LIN {X 0,Y 353.658,Z 542.313,A -85,B 0,C 180,E1 -13402.004,E2 -13402.004} C_VEL
LIN {X 0,Y 353.447,Z 546.534,A -85,B 0,C 180,E1 -13403.832,E2 -13403.832} C_VEL
LIN {X 0,Y 353.361,Z 549.292,A -85,B 0,C 180,E1 -13405.437,E2 -13405.437} C_VEL
LIN {X 0,Y 353.332,Z 551.715,A -85,B 0,C 180,E1 -13407.72,E2 -13407.72} C_VEL
LIN {X 0,Y 353.402,Z 552.336,A -85,B 0,C 180,E1 -13408.86,E2 -13408.86} C_VEL
LIN {X 0,Y 353.411,Z 552.555,A -85,B 0,C 180,E1 -13410,E2 -13410} C_VEL
LIN {X 0,Y 353.42,Z 552.336,A -85,B 0,C 180,E1 -13411.139,E2 -13411.139} C_VEL
LIN {X 0,Y 353.332,Z 551.714,A -85,B 0,C 180,E1 -13412.28,E2 -13412.28} C_VEL
LIN {X 0,Y 353.36,Z 549.289,A -85,B 0,C 180,E1 -13414.563,E2 -13414.563} C_VEL
LIN {X 0,Y 353.446,Z 546.529,A -85,B 0,C 180,E1 -13416.167,E2 -13416.167} C_VEL
LIN {X 0,Y 353.653,Z 542.299,A -85,B 0,C 180,E1 -13417.996,E2 -13417.996} C_VEL
LIN {X 0,Y 354.203,Z 536.136,A -85,B 0,C 180,E1 -13419.998,E2 -13419.998} C_VEL
LIN {X 0,Y 354.809,Z 529.405,A -85,B 0,C 180,E1 -13421.714,E2 -13421.714} C_VEL
LIN {X 0,Y 355.835,Z 521.078,A -85,B 0,C 180,E1 -13423.419,E2 -13423.419} C_VEL
LIN {X 0,Y 356.804,Z 512.544,A -85,B 0,C 180,E1 -13424.837,E2 -13424.837} C_VEL
LIN {X 0,Y 357.663,Z 503.178,A -85,B 0,C 180,E1 -13426.114,E2 -13426.114} C_VEL
LIN {X 0,Y 358.907,Z 491.587,A -85,B 0,C 180,E1 -13427.375,E2 -13427.375} C_VEL
LIN {X 0,Y 359.729,Z 483.732,A -85,B 0,C 180,E1 -13428.068,E2 -13428.068} C_VEL
LIN {X 0,Y 358.634,Z 471.661,A -85,B 0,C 180,E1 -13429.025,E2 -13429.025} C_VEL
LIN {X 0,Y 356.865,Z 458.288,A -85,B 0,C 180,E1 -13429.859,E2 -13429.859} C_VEL
LIN {X 0,Y 354.4,Z 444.565,A -85,B 0,C 180,E1 -13430.496,E2 -13430.496} C_VEL
LIN {X 0,Y 354.928,Z 437.738,A -85,B 0,C 180,E1 -13433.871,E2 -13433.871} C_VEL
LIN {X 0,Y 355.677,Z 429.964,A -85,B 0,C 180,E1 -13437.687,E2 -13437.687} C_VEL
LIN {X 0,Y 356.481,Z 422.367,A -85,B 0,C 180,E1 -13441.46,E2 -13441.46} C_VEL
LIN {X 0,Y 357.26,Z 415.856,A -85,B 0,C 180,E1 -13444.784,E2 -13444.784} C_VEL
LIN {X 0,Y 357.465,Z 411.958,A -85,B 0,C 180,E1 -13446.86,E2 -13446.86} C_VEL
LIN {X 0,Y 356.763,Z 406.874,A -85,B 0,C 180,E1 -13449.801,E2 -13449.801} C_VEL
LIN {X 0,Y 355.812,Z 401.617,A -85,B 0,C 180,E1 -13453.044,E2 -13453.044} C_VEL
LIN {X 0,Y 354.813,Z 396.295,A -85,B 0,C 180,E1 -13456.602,E2 -13456.602} C_VEL
LIN {X 0,Y 354.817,Z 396.29,A -85,B 0,C 180,E1 -13460.666,E2 -13460.666} C_VEL
LIN {X 0,Y 354.824,Z 396.285,A -85,B 0,C 180,E1 -13464.301,E2 -13464.301} C_VEL
LIN {X 0,Y 354.79,Z 396.288,A -85,B 0,C 180,E1 -13467.667,E2 -13467.667} C_VEL
LIN {X 0,Y 354.848,Z 396.28,A -85,B 0,C 180,E1 -13471.619,E2 -13471.619} C_VEL
LIN {X 0,Y 354.901,Z 396.275,A -85,B 0,C 180,E1 -13474.173,E2 -13474.173} C_VEL
LIN {X 0,Y 354.837,Z 396.282,A -85,B 0,C 180,E1 -13477.894,E2 -13477.894} C_VEL
LIN {X 0,Y 354.925,Z 396.271,A -85,B 0,C 180,E1 -13481.892,E2 -13481.892} C_VEL
LIN {X 0,Y 354.946,Z 396.269,A -85,B 0,C 180,E1 -13485.981,E2 -13485.981} C_VEL
LIN {X 0,Y 354.986,Z 396.263,A -85,B 0,C 180,E1 -13489.736,E2 -13489.736} C_VEL
LIN {X 0,Y 355.118,Z 396.249,A -85,B 0,C 180,E1 -13492.037,E2 -13492.037} C_VEL
LIN {X 0,Y 355.095,Z 396.255,A -85,B 0,C 180,E1 -13494.321,E2 -13494.321} C_VEL
LIN {X 0,Y 355.247,Z 396.231,A -85,B 0,C 180,E1 -13497.732,E2 -13497.732} C_VEL
LIN {X 0,Y 355.401,Z 396.214,A -85,B 0,C 180,E1 -13500,E2 -13500} C_VEL
LIN {X 0,Y 355.247,Z 396.236,A -85,B 0,C 180,E1 -13502.268,E2 -13502.268} C_VEL
LIN {X 0,Y 355.142,Z 396.245,A -85,B 0,C 180,E1 -13506.819,E2 -13506.819} C_VEL
LIN {X 0,Y 355.018,Z 396.259,A -85,B 0,C 180,E1 -13509.112,E2 -13509.112} C_VEL
LIN {X 0,Y 354.924,Z 396.273,A -85,B 0,C 180,E1 -13512.581,E2 -13512.581} C_VEL
LIN {X 0,Y 354.893,Z 396.281,A -85,B 0,C 180,E1 -13516.096,E2 -13516.096} C_VEL
LIN {X 0,Y 354.906,Z 396.275,A -85,B 0,C 180,E1 -13518.472,E2 -13518.472} C_VEL
LIN {X 0,Y 354.829,Z 396.288,A -85,B 0,C 180,E1 -13522.107,E2 -13522.107} C_VEL
LIN {X 0,Y 354.901,Z 396.278,A -85,B 0,C 180,E1 -13525.827,E2 -13525.827} C_VEL
LIN {X 0,Y 354.82,Z 396.287,A -85,B 0,C 180,E1 -13529.682,E2 -13529.682} C_VEL
LIN {X 0,Y 354.808,Z 396.289,A -85,B 0,C 180,E1 -13533.702,E2 -13533.702} C_VEL
LIN {X 0,Y 354.804,Z 396.286,A -85,B 0,C 180,E1 -13536.459,E2 -13536.459} C_VEL
LIN {X 0,Y 354.826,Z 396.286,A -85,B 0,C 180,E1 -13539.424,E2 -13539.424} C_VEL
LIN {X 0,Y 354.793,Z 396.287,A -85,B 0,C 180,E1 -13542.868,E2 -13542.868} C_VEL
LIN {X 0,Y 354.854,Z 396.281,A -85,B 0,C 180,E1 -13546.117,E2 -13546.117} C_VEL
LIN {X 0,Y 354.859,Z 396.281,A -85,B 0,C 180,E1 -13549.189,E2 -13549.189} C_VEL
LIN {X 0,Y 354.792,Z 396.288,A -85,B 0,C 180,E1 -13552.406,E2 -13552.406} C_VEL
LIN {X 0,Y 354.649,Z 396.307,A -85,B 0,C 180,E1 -13554.922,E2 -13554.922} C_VEL
LIN {X 0,Y 354.269,Z 396.37,A -85,B 0,C 180,E1 -13558.544,E2 -13558.544} C_VEL
LIN {X 0,Y 354.19,Z 398.943,A -85,B 0,C 180,E1 -13561.561,E2 -13561.561} C_VEL
LIN {X 0,Y 354.109,Z 401.198,A -85,B 0,C 180,E1 -13564.111,E2 -13564.111} C_VEL
LIN {X 0,Y 354.046,Z 403.503,A -85,B 0,C 180,E1 -13566.609,E2 -13566.609} C_VEL
LIN {X 0,Y 354.017,Z 406.555,A -85,B 0,C 180,E1 -13569.603,E2 -13569.603} C_VEL
LIN {X 0,Y 357.841,Z 419.612,A -85,B 0,C 180,E1 -13570.357,E2 -13570.357} C_VEL
LIN {X 0,Y 360.654,Z 431.525,A -85,B 0,C 180,E1 -13571.219,E2 -13571.219} C_VEL
LIN {X 0,Y 361.301,Z 435.514,A -85,B 0,C 180,E1 -13571.542,E2 -13571.542} C_VEL
LIN {X 0,Y 360.301,Z 447.888,A -85,B 0,C 180,E1 -13572.548,E2 -13572.548} C_VEL
LIN {X 0,Y 359.4,Z 458.522,A -85,B 0,C 180,E1 -13573.674,E2 -13573.674} C_VEL
LIN {X 0,Y 358.359,Z 468.201,A -85,B 0,C 180,E1 -13574.939,E2 -13574.939} C_VEL
LIN {X 0,Y 357.248,Z 477.008,A -85,B 0,C 180,E1 -13576.345,E2 -13576.345} C_VEL
LIN {X 0,Y 356.228,Z 485.588,A -85,B 0,C 180,E1 -13578.044,E2 -13578.044} C_VEL
LIN {X 0,Y 355.358,Z 492.423,A -85,B 0,C 180,E1 -13579.747,E2 -13579.747} C_VEL
LIN {X 0,Y 354.706,Z 497.89,A -85,B 0,C 180,E1 -13581.454,E2 -13581.454} C_VEL
LIN {X 0,Y 354.252,Z 502.177,A -85,B 0,C 180,E1 -13583.164,E2 -13583.164} C_VEL
LIN {X 0,Y 353.919,Z 504.45,A -85,B 0,C 180,E1 -13584.302,E2 -13584.302} C_VEL
LIN {X 0,Y 353.78,Z 506.291,A -85,B 0,C 180,E1 -13585.442,E2 -13585.442} C_VEL
LIN {X 0,Y 353.784,Z 507.67,A -85,B 0,C 180,E1 -13586.583,E2 -13586.583} C_VEL
LIN {X 0,Y 353.508,Z 509.272,A -85,B 0,C 180,E1 -13588.861,E2 -13588.861} C_VEL
LIN {X 0,Y 353.477,Z 509.503,A -85,B 0,C 180,E1 -13590,E2 -13590} C_VEL
LIN {X 0,Y 353.636,Z 508.728,A -85,B 0,C 180,E1 -13592.278,E2 -13592.278} C_VEL
LIN {X 0,Y 353.764,Z 507.766,A -85,B 0,C 180,E1 -13593.417,E2 -13593.417} C_VEL
LIN {X 0,Y 353.777,Z 506.428,A -85,B 0,C 180,E1 -13594.558,E2 -13594.558} C_VEL
LIN {X 0,Y 354.082,Z 503.581,A -85,B 0,C 180,E1 -13596.267,E2 -13596.267} C_VEL
LIN {X 0,Y 354.483,Z 499.722,A -85,B 0,C 180,E1 -13597.978,E2 -13597.978} C_VEL
LIN {X 0,Y 355.096,Z 494.736,A -85,B 0,C 180,E1 -13599.685,E2 -13599.685} C_VEL
LIN {X 0,Y 355.914,Z 488.452,A -85,B 0,C 180,E1 -13601.389,E2 -13601.389} C_VEL
LIN {X 0,Y 356.891,Z 480.584,A -85,B 0,C 180,E1 -13603.089,E2 -13603.089} C_VEL
LIN {X 0,Y 357.857,Z 472.558,A -85,B 0,C 180,E1 -13604.501,E2 -13604.501} C_VEL
LIN {X 0,Y 358.974,Z 462.756,A -85,B 0,C 180,E1 -13605.908,E2 -13605.908} C_VEL
LIN {X 0,Y 359.828,Z 453.112,A -85,B 0,C 180,E1 -13607.036,E2 -13607.036} C_VEL
LIN {X 0,Y 360.762,Z 442.655,A -85,B 0,C 180,E1 -13608.015,E2 -13608.015} C_VEL
LIN {X 0,Y 361.217,Z 433.881,A -85,B 0,C 180,E1 -13608.687,E2 -13608.687} C_VEL
LIN {X 0,Y 358.725,Z 422.991,A -85,B 0,C 180,E1 -13609.522,E2 -13609.522} C_VEL
LIN {X 0,Y 355.128,Z 410.483,A -85,B 0,C 180,E1 -13610.301,E2 -13610.301} C_VEL
LIN {X 0,Y 353.959,Z 406.397,A -85,B 0,C 180,E1 -13610.514,E2 -13610.514} C_VEL
LIN {X 0,Y 354.101,Z 402.965,A -85,B 0,C 180,E1 -13614.078,E2 -13614.078} C_VEL
LIN {X 0,Y 354.141,Z 400.17,A -85,B 0,C 180,E1 -13617.158,E2 -13617.158} C_VEL
LIN {X 0,Y 354.258,Z 397.914,A -85,B 0,C 180,E1 -13619.734,E2 -13619.734} C_VEL
LIN {X 0,Y 354.3,Z 396.464,A -85,B 0,C 180,E1 -13621.464,E2 -13621.464} C_VEL
LIN {X 0,Y 354.651,Z 396.307,A -85,B 0,C 180,E1 -13625.078,E2 -13625.078} C_VEL
LIN {X 0,Y 354.769,Z 396.29,A -85,B 0,C 180,E1 -13627.355,E2 -13627.355} C_VEL
LIN {X 0,Y 354.164,Z 396.37,A -85,B 0,C 180,E1 -13628.302,E2 -13628.302} C_VEL
LIN {X 0,Y 351.329,Z 396.72,A -85,B 0,C 180,E1 -13629.843,E2 -13629.843} C_VEL
LIN {X 0,Y 348.879,Z 397.025,A -85,B 0,C 180,E1 -13631.09,E2 -13631.09} C_VEL
LIN {X 0,Y 347.811,Z 397.159,A -85,B 0,C 180,E1 -13632.055,E2 -13632.055} C_VEL
LIN {X 0,Y 347.717,Z 397.166,A -85,B 0,C 180,E1 -13632.382,E2 -13632.382} C_VEL
LIN {X 0,Y 347.709,Z 397.17,A -85,B 0,C 180,E1 -13635.027,E2 -13635.027} C_VEL
LIN {X 0,Y 347.754,Z 397.17,A -85,B 0,C 180,E1 -13638.397,E2 -13638.397} C_VEL
LIN {X 0,Y 347.781,Z 397.164,A -85,B 0,C 180,E1 -13642.011,E2 -13642.011} C_VEL
LIN {X 0,Y 347.748,Z 397.165,A -85,B 0,C 180,E1 -13645.536,E2 -13645.536} C_VEL
LIN {X 0,Y 347.749,Z 397.17,A -85,B 0,C 180,E1 -13648.301,E2 -13648.301} C_VEL
LIN {X 0,Y 347.782,Z 397.161,A -85,B 0,C 180,E1 -13650.988,E2 -13650.988} C_VEL
LIN {X 0,Y 347.834,Z 397.156,A -85,B 0,C 180,E1 -13653.608,E2 -13653.608} C_VEL
LIN {X 0,Y 347.789,Z 397.165,A -85,B 0,C 180,E1 -13656.162,E2 -13656.162} C_VEL
LIN {X 0,Y 347.813,Z 397.162,A -85,B 0,C 180,E1 -13659.909,E2 -13659.909} C_VEL
LIN {X 0,Y 347.87,Z 397.152,A -85,B 0,C 180,E1 -13662.359,E2 -13662.359} C_VEL
LIN {X 0,Y 347.901,Z 397.151,A -85,B 0,C 180,E1 -13665.971,E2 -13665.971} C_VEL
LIN {X 0,Y 347.931,Z 397.145,A -85,B 0,C 180,E1 -13669.526,E2 -13669.526} C_VEL
LIN {X 0,Y 348.084,Z 397.123,A -85,B 0,C 180,E1 -13673.042,E2 -13673.042} C_VEL
LIN {X 0,Y 348.21,Z 397.113,A -85,B 0,C 180,E1 -13677.686,E2 -13677.686} C_VEL
LIN {X 0,Y 348.349,Z 397.093,A -85,B 0,C 180,E1 -13680,E2 -13680} C_VEL
LIN {X 0,Y 348.21,Z 397.108,A -85,B 0,C 180,E1 -13682.313,E2 -13682.313} C_VEL
LIN {X 0,Y 348.111,Z 397.12,A -85,B 0,C 180,E1 -13686.958,E2 -13686.958} C_VEL
LIN {X 0,Y 347.973,Z 397.14,A -85,B 0,C 180,E1 -13689.298,E2 -13689.298} C_VEL
LIN {X 0,Y 347.898,Z 397.147,A -85,B 0,C 180,E1 -13692.839,E2 -13692.839} C_VEL
LIN {X 0,Y 347.843,Z 397.153,A -85,B 0,C 180,E1 -13696.431,E2 -13696.431} C_VEL
LIN {X 0,Y 347.855,Z 397.153,A -85,B 0,C 180,E1 -13698.86,E2 -13698.86} C_VEL
LIN {X 0,Y 347.778,Z 397.161,A -85,B 0,C 180,E1 -13702.579,E2 -13702.579} C_VEL
LIN {X 0,Y 347.816,Z 397.161,A -85,B 0,C 180,E1 -13705.108,E2 -13705.108} C_VEL
LIN {X 0,Y 347.811,Z 397.159,A -85,B 0,C 180,E1 -13707.694,E2 -13707.694} C_VEL
LIN {X 0,Y 347.752,Z 397.165,A -85,B 0,C 180,E1 -13710.348,E2 -13710.348} C_VEL
LIN {X 0,Y 347.751,Z 397.165,A -85,B 0,C 180,E1 -13714.044,E2 -13714.044} C_VEL
LIN {X 0,Y 347.765,Z 397.167,A -85,B 0,C 180,E1 -13717.32,E2 -13717.32} C_VEL
LIN {X 0,Y 347.735,Z 397.169,A -85,B 0,C 180,E1 -13720.297,E2 -13720.297} C_VEL
LIN {X 0,Y 347.773,Z 397.235,A -85,B 0,C 180,E1 -13722.971,E2 -13722.971} C_VEL
LIN {X 0,Y 348.737,Z 402.423,A -85,B 0,C 180,E1 -13726.511,E2 -13726.511} C_VEL
LIN {X 0,Y 349.739,Z 407.928,A -85,B 0,C 180,E1 -13729.981,E2 -13729.981} C_VEL
LIN {X 0,Y 350.471,Z 413.076,A -85,B 0,C 180,E1 -13733.016,E2 -13733.016} C_VEL
LIN {X 0,Y 350.197,Z 417.38,A -85,B 0,C 180,E1 -13735.368,E2 -13735.368} C_VEL
LIN {X 0,Y 349.43,Z 423.299,A -85,B 0,C 180,E1 -13738.471,E2 -13738.471} C_VEL
LIN {X 0,Y 348.601,Z 430.928,A -85,B 0,C 180,E1 -13742.374,E2 -13742.374} C_VEL
LIN {X 0,Y 347.838,Z 438.435,A -85,B 0,C 180,E1 -13746.165,E2 -13746.165} C_VEL
LIN {X 0,Y 347.377,Z 444.195,A -85,B 0,C 180,E1 -13749.071,E2 -13749.071} C_VEL
LIN {X 0,Y 349.885,Z 457.827,A -85,B 0,C 180,E1 -13749.719,E2 -13749.719} C_VEL
LIN {X 0,Y 351.588,Z 470.563,A -85,B 0,C 180,E1 -13750.528,E2 -13750.528} C_VEL
LIN {X 0,Y 352.829,Z 483.366,A -85,B 0,C 180,E1 -13751.566,E2 -13751.566} C_VEL
LIN {X 0,Y 351.846,Z 494.074,A -85,B 0,C 180,E1 -13752.565,E2 -13752.565} C_VEL
LIN {X 0,Y 350.581,Z 505.021,A -85,B 0,C 180,E1 -13753.851,E2 -13753.851} C_VEL
LIN {X 0,Y 349.688,Z 513.954,A -85,B 0,C 180,E1 -13755.152,E2 -13755.152} C_VEL
LIN {X 0,Y 348.731,Z 522.173,A -85,B 0,C 180,E1 -13756.599,E2 -13756.599} C_VEL
LIN {X 0,Y 347.667,Z 530.237,A -85,B 0,C 180,E1 -13758.337,E2 -13758.337} C_VEL
LIN {X 0,Y 347.071,Z 536.725,A -85,B 0,C 180,E1 -13760.089,E2 -13760.089} C_VEL
LIN {X 0,Y 346.595,Z 541.879,A -85,B 0,C 180,E1 -13761.84,E2 -13761.84} C_VEL
LIN {X 0,Y 346.344,Z 546.435,A -85,B 0,C 180,E1 -13763.885,E2 -13763.885} C_VEL
LIN {X 0,Y 346.275,Z 548.86,A -85,B 0,C 180,E1 -13765.343,E2 -13765.343} C_VEL
LIN {X 0,Y 346.237,Z 551.283,A -85,B 0,C 180,E1 -13767.673,E2 -13767.673} C_VEL
LIN {X 0,Y 346.322,Z 551.905,A -85,B 0,C 180,E1 -13768.837,E2 -13768.837} C_VEL
LIN {X 0,Y 346.35,Z 552.125,A -85,B 0,C 180,E1 -13770,E2 -13770} C_VEL
LIN {X 0,Y 346.339,Z 551.904,A -85,B 0,C 180,E1 -13771.163,E2 -13771.163} C_VEL
LIN {X 0,Y 346.206,Z 550.269,A -85,B 0,C 180,E1 -13773.491,E2 -13773.491} C_VEL
LIN {X 0,Y 346.274,Z 548.856,A -85,B 0,C 180,E1 -13774.657,E2 -13774.657} C_VEL
LIN {X 0,Y 346.343,Z 546.429,A -85,B 0,C 180,E1 -13776.113,E2 -13776.113} C_VEL
LIN {X 0,Y 346.591,Z 541.863,A -85,B 0,C 180,E1 -13778.16,E2 -13778.16} C_VEL
LIN {X 0,Y 347.171,Z 535.699,A -85,B 0,C 180,E1 -13780.203,E2 -13780.203} C_VEL
LIN {X 0,Y 347.819,Z 528.968,A -85,B 0,C 180,E1 -13781.953,E2 -13781.953} C_VEL
LIN {X 0,Y 348.865,Z 520.639,A -85,B 0,C 180,E1 -13783.692,E2 -13783.692} C_VEL
LIN {X 0,Y 349.932,Z 511.43,A -85,B 0,C 180,E1 -13785.238,E2 -13785.238} C_VEL
LIN {X 0,Y 350.949,Z 501.56,A -85,B 0,C 180,E1 -13786.581,E2 -13786.581} C_VEL
LIN {X 0,Y 352.282,Z 489.717,A -85,B 0,C 180,E1 -13787.862,E2 -13787.862} C_VEL
LIN {X 0,Y 352.82,Z 483.284,A -85,B 0,C 180,E1 -13788.435,E2 -13788.435} C_VEL
LIN {X 0,Y 351.587,Z 470.464,A -85,B 0,C 180,E1 -13789.47,E2 -13789.47} C_VEL
LIN {X 0,Y 349.733,Z 457.055,A -85,B 0,C 180,E1 -13790.316,E2 -13790.316} C_VEL
LIN {X 0,Y 347.391,Z 444.134,A -85,B 0,C 180,E1 -13790.919,E2 -13790.919} C_VEL
LIN {X 0,Y 348.085,Z 435.921,A -85,B 0,C 180,E1 -13795.087,E2 -13795.087} C_VEL
LIN {X 0,Y 348.873,Z 428.36,A -85,B 0,C 180,E1 -13798.913,E2 -13798.913} C_VEL
LIN {X 0,Y 349.762,Z 420.671,A -85,B 0,C 180,E1 -13802.856,E2 -13802.856} C_VEL
LIN {X 0,Y 350.378,Z 415.533,A -85,B 0,C 180,E1 -13805.57,E2 -13805.57} C_VEL
LIN {X 0,Y 350.334,Z 411.671,A -85,B 0,C 180,E1 -13807.724,E2 -13807.724} C_VEL
LIN {X 0,Y 349.526,Z 406.519,A -85,B 0,C 180,E1 -13810.835,E2 -13810.835} C_VEL
LIN {X 0,Y 348.533,Z 401.184,A -85,B 0,C 180,E1 -13814.279,E2 -13814.279} C_VEL
LIN {X 0,Y 347.75,Z 397.175,A -85,B 0,C 180,E1 -13817.122,E2 -13817.122} C_VEL
LIN {X 0,Y 347.754,Z 397.168,A -85,B 0,C 180,E1 -13821.208,E2 -13821.208} C_VEL
LIN {X 0,Y 347.791,Z 397.16,A -85,B 0,C 180,E1 -13824.125,E2 -13824.125} C_VEL
LIN {X 0,Y 347.741,Z 397.167,A -85,B 0,C 180,E1 -13828.086,E2 -13828.086} C_VEL
LIN {X 0,Y 347.781,Z 397.165,A -85,B 0,C 180,E1 -13830.988,E2 -13830.988} C_VEL
LIN {X 0,Y 347.833,Z 397.154,A -85,B 0,C 180,E1 -13833.608,E2 -13833.608} C_VEL
LIN {X 0,Y 347.791,Z 397.161,A -85,B 0,C 180,E1 -13836.162,E2 -13836.162} C_VEL
LIN {X 0,Y 347.815,Z 397.157,A -85,B 0,C 180,E1 -13839.909,E2 -13839.909} C_VEL
LIN {X 0,Y 347.869,Z 397.153,A -85,B 0,C 180,E1 -13842.359,E2 -13842.359} C_VEL
LIN {X 0,Y 347.9,Z 397.147,A -85,B 0,C 180,E1 -13845.971,E2 -13845.971} C_VEL
LIN {X 0,Y 347.936,Z 397.141,A -85,B 0,C 180,E1 -13849.526,E2 -13849.526} C_VEL
LIN {X 0,Y 348.078,Z 397.125,A -85,B 0,C 180,E1 -13851.875,E2 -13851.875} C_VEL
LIN {X 0,Y 348.07,Z 397.129,A -85,B 0,C 180,E1 -13854.206,E2 -13854.206} C_VEL
LIN {X 0,Y 348.209,Z 397.108,A -85,B 0,C 180,E1 -13857.687,E2 -13857.687} C_VEL
LIN {X 0,Y 348.371,Z 397.09,A -85,B 0,C 180,E1 -13860,E2 -13860} C_VEL
LIN {X 0,Y 348.209,Z 397.113,A -85,B 0,C 180,E1 -13862.314,E2 -13862.314} C_VEL
LIN {X 0,Y 348.11,Z 397.12,A -85,B 0,C 180,E1 -13866.958,E2 -13866.958} C_VEL
LIN {X 0,Y 347.97,Z 397.137,A -85,B 0,C 180,E1 -13869.299,E2 -13869.299} C_VEL
LIN {X 0,Y 347.893,Z 397.147,A -85,B 0,C 180,E1 -13872.839,E2 -13872.839} C_VEL
LIN {X 0,Y 347.842,Z 397.156,A -85,B 0,C 180,E1 -13876.431,E2 -13876.431} C_VEL
LIN {X 0,Y 347.855,Z 397.151,A -85,B 0,C 180,E1 -13878.86,E2 -13878.86} C_VEL
LIN {X 0,Y 347.771,Z 397.163,A -85,B 0,C 180,E1 -13882.58,E2 -13882.58} C_VEL
LIN {X 0,Y 347.813,Z 397.157,A -85,B 0,C 180,E1 -13885.108,E2 -13885.108} C_VEL
LIN {X 0,Y 347.811,Z 397.16,A -85,B 0,C 180,E1 -13887.694,E2 -13887.694} C_VEL
LIN {X 0,Y 347.751,Z 397.166,A -85,B 0,C 180,E1 -13890.348,E2 -13890.348} C_VEL
LIN {X 0,Y 347.75,Z 397.169,A -85,B 0,C 180,E1 -13894.044,E2 -13894.044} C_VEL
LIN {X 0,Y 347.768,Z 397.163,A -85,B 0,C 180,E1 -13897.32,E2 -13897.32} C_VEL
LIN {X 0,Y 347.735,Z 397.168,A -85,B 0,C 180,E1 -13900.297,E2 -13900.297} C_VEL
LIN {X 0,Y 347.731,Z 397.17,A -85,B 0,C 180,E1 -13903.407,E2 -13903.407} C_VEL
LIN {X 0,Y 347.788,Z 397.16,A -85,B 0,C 180,E1 -13906.676,E2 -13906.676} C_VEL
LIN {X 0,Y 347.788,Z 397.161,A -85,B 0,C 180,E1 -13910.165,E2 -13910.165} C_VEL
LIN {X 0,Y 347.739,Z 397.167,A -85,B 0,C 180,E1 -13912.676,E2 -13912.676} C_VEL
LIN {X 0,Y 347.491,Z 397.202,A -85,B 0,C 180,E1 -13916.02,E2 -13916.02} C_VEL
LIN {X 0,Y 347.269,Z 397.229,A -85,B 0,C 180,E1 -13918.252,E2 -13918.252} C_VEL
LIN {X 0,Y 347.183,Z 399.317,A -85,B 0,C 180,E1 -13920.933,E2 -13920.933} C_VEL
LIN {X 0,Y 347.093,Z 401.598,A -85,B 0,C 180,E1 -13923.547,E2 -13923.547} C_VEL
LIN {X 0,Y 347.043,Z 403.914,A -85,B 0,C 180,E1 -13926.107,E2 -13926.107} C_VEL
LIN {X 0,Y 346.988,Z 406.939,A -85,B 0,C 180,E1 -13929.168,E2 -13929.168} C_VEL
LIN {X 0,Y 350.853,Z 420.05,A -85,B 0,C 180,E1 -13929.948,E2 -13929.948} C_VEL
LIN {X 0,Y 353.848,Z 432.487,A -85,B 0,C 180,E1 -13930.878,E2 -13930.878} C_VEL
LIN {X 0,Y 354.574,Z 436.195,A -85,B 0,C 180,E1 -13931.198,E2 -13931.198} C_VEL
LIN {X 0,Y 353.563,Z 448.324,A -85,B 0,C 180,E1 -13932.205,E2 -13932.205} C_VEL
LIN {X 0,Y 352.559,Z 459.427,A -85,B 0,C 180,E1 -13933.409,E2 -13933.409} C_VEL
LIN {X 0,Y 351.531,Z 468.635,A -85,B 0,C 180,E1 -13934.639,E2 -13934.639} C_VEL
LIN {X 0,Y 350.362,Z 477.443,A -85,B 0,C 180,E1 -13936.072,E2 -13936.072} C_VEL
LIN {X 0,Y 349.304,Z 486.021,A -85,B 0,C 180,E1 -13937.804,E2 -13937.804} C_VEL
LIN {X 0,Y 348.396,Z 492.856,A -85,B 0,C 180,E1 -13939.54,E2 -13939.54} C_VEL
LIN {X 0,Y 347.693,Z 498.324,A -85,B 0,C 180,E1 -13941.28,E2 -13941.28} C_VEL
LIN {X 0,Y 347.212,Z 502.61,A -85,B 0,C 180,E1 -13943.024,E2 -13943.024} C_VEL
LIN {X 0,Y 346.885,Z 504.882,A -85,B 0,C 180,E1 -13944.186,E2 -13944.186} C_VEL
LIN {X 0,Y 346.707,Z 506.724,A -85,B 0,C 180,E1 -13945.349,E2 -13945.349} C_VEL
LIN {X 0,Y 346.713,Z 508.102,A -85,B 0,C 180,E1 -13946.514,E2 -13946.514} C_VEL
LIN {X 0,Y 346.583,Z 509.09,A -85,B 0,C 180,E1 -13947.676,E2 -13947.676} C_VEL
LIN {X 0,Y 346.413,Z 509.933,A -85,B 0,C 180,E1 -13950,E2 -13950} C_VEL
LIN {X 0,Y 346.58,Z 509.158,A -85,B 0,C 180,E1 -13952.324,E2 -13952.324} C_VEL
LIN {X 0,Y 346.695,Z 508.197,A -85,B 0,C 180,E1 -13953.487,E2 -13953.487} C_VEL
LIN {X 0,Y 346.705,Z 506.859,A -85,B 0,C 180,E1 -13954.651,E2 -13954.651} C_VEL
LIN {X 0,Y 347.059,Z 504.011,A -85,B 0,C 180,E1 -13956.395,E2 -13956.395} C_VEL
LIN {X 0,Y 347.467,Z 500.152,A -85,B 0,C 180,E1 -13958.14,E2 -13958.14} C_VEL
LIN {X 0,Y 348.099,Z 495.167,A -85,B 0,C 180,E1 -13959.882,E2 -13959.882} C_VEL
LIN {X 0,Y 348.965,Z 488.882,A -85,B 0,C 180,E1 -13961.619,E2 -13961.619} C_VEL
LIN {X 0,Y 350.002,Z 481.012,A -85,B 0,C 180,E1 -13963.351,E2 -13963.351} C_VEL
LIN {X 0,Y 351.013,Z 472.985,A -85,B 0,C 180,E1 -13964.79,E2 -13964.79} C_VEL
LIN {X 0,Y 352.165,Z 463.183,A -85,B 0,C 180,E1 -13966.224,E2 -13966.224} C_VEL
LIN {X 0,Y 353.067,Z 453.538,A -85,B 0,C 180,E1 -13967.373,E2 -13967.373} C_VEL
LIN {X 0,Y 354.05,Z 443.078,A -85,B 0,C 180,E1 -13968.369,E2 -13968.369} C_VEL
LIN {X 0,Y 354.548,Z 435.819,A -85,B 0,C 180,E1 -13968.937,E2 -13968.937} C_VEL
LIN {X 0,Y 352.026,Z 424.588,A -85,B 0,C 180,E1 -13969.84,E2 -13969.84} C_VEL
LIN {X 0,Y 348.492,Z 412.001,A -85,B 0,C 180,E1 -13970.667,E2 -13970.667} C_VEL
LIN {X 0,Y 346.913,Z 406.812,A -85,B 0,C 180,E1 -13970.969,E2 -13970.969} C_VEL
LIN {X 0,Y 347.042,Z 403.633,A -85,B 0,C 180,E1 -13974.313,E2 -13974.313} C_VEL
LIN {X 0,Y 347.105,Z 400.558,A -85,B 0,C 180,E1 -13977.755,E2 -13977.755} C_VEL
LIN {X 0,Y 347.221,Z 398.286,A -85,B 0,C 180,E1 -13980.399,E2 -13980.399} C_VEL
LIN {X 0,Y 347.273,Z 397.23,A -85,B 0,C 180,E1 -13981.79,E2 -13981.79} C_VEL
LIN {X 0,Y 347.556,Z 397.195,A -85,B 0,C 180,E1 -13984.486,E2 -13984.486} C_VEL
LIN {X 0,Y 347.766,Z 397.164,A -85,B 0,C 180,E1 -13987.987,E2 -13987.987} C_VEL
LIN {X 0,Y 347.754,Z 397.165,A -85,B 0,C 180,E1 -13991.83,E2 -13991.83} C_VEL
LIN {X 0,Y 347.717,Z 397.166,A -85,B 0,C 180,E1 -13992.382,E2 -13992.382} C_VEL
LIN {X 0,Y 347.029,Z 397.255,A -85,B 0,C 180,E1 -13993.349,E2 -13993.349} C_VEL
LIN {X 0,Y 344.166,Z 397.612,A -85,B 0,C 180,E1 -13994.921,E2 -13994.921} C_VEL
LIN {X 0,Y 341.765,Z 397.914,A -85,B 0,C 180,E1 -13996.194,E2 -13996.194} C_VEL
LIN {X 0,Y 340.754,Z 398.036,A -85,B 0,C 180,E1 -13997.18,E2 -13997.18} C_VEL
LIN {X 0,Y 340.681,Z 398.045,A -85,B 0,C 180,E1 -13997.513,E2 -13997.513} C_VEL
LIN {X 0,Y 340.703,Z 398.048,A -85,B 0,C 180,E1 -14000.248,E2 -14000.248} C_VEL
LIN {X 0,Y 340.715,Z 398.041,A -85,B 0,C 180,E1 -14003.559,E2 -14003.559} C_VEL
LIN {X 0,Y 340.698,Z 398.048,A -85,B 0,C 180,E1 -14006.154,E2 -14006.154} C_VEL
LIN {X 0,Y 340.745,Z 398.041,A -85,B 0,C 180,E1 -14010.329,E2 -14010.329} C_VEL
LIN {X 0,Y 340.807,Z 398.029,A -85,B 0,C 180,E1 -14013.02,E2 -14013.02} C_VEL
LIN {X 0,Y 340.758,Z 398.037,A -85,B 0,C 180,E1 -14015.638,E2 -14015.638} C_VEL
LIN {X 0,Y 340.739,Z 398.039,A -85,B 0,C 180,E1 -14019.474,E2 -14019.474} C_VEL
LIN {X 0,Y 340.862,Z 398.029,A -85,B 0,C 180,E1 -14021.984,E2 -14021.984} C_VEL
LIN {X 0,Y 340.873,Z 398.025,A -85,B 0,C 180,E1 -14025.705,E2 -14025.705} C_VEL
LIN {X 0,Y 340.874,Z 398.022,A -85,B 0,C 180,E1 -14029.306,E2 -14029.306} C_VEL
LIN {X 0,Y 341.051,Z 397.999,A -85,B 0,C 180,E1 -14032.898,E2 -14032.898} C_VEL
LIN {X 0,Y 341.172,Z 397.99,A -85,B 0,C 180,E1 -14037.639,E2 -14037.639} C_VEL
LIN {X 0,Y 341.299,Z 397.972,A -85,B 0,C 180,E1 -14040,E2 -14040} C_VEL
LIN {X 0,Y 341.172,Z 397.985,A -85,B 0,C 180,E1 -14042.361,E2 -14042.361} C_VEL
LIN {X 0,Y 341.081,Z 397.997,A -85,B 0,C 180,E1 -14047.102,E2 -14047.102} C_VEL
LIN {X 0,Y 340.88,Z 398.021,A -85,B 0,C 180,E1 -14050.693,E2 -14050.693} C_VEL
LIN {X 0,Y 340.867,Z 398.022,A -85,B 0,C 180,E1 -14054.325,E2 -14054.325} C_VEL
LIN {X 0,Y 340.841,Z 398.025,A -85,B 0,C 180,E1 -14058.466,E2 -14058.466} C_VEL
LIN {X 0,Y 340.757,Z 398.037,A -85,B 0,C 180,E1 -14061.857,E2 -14061.857} C_VEL
LIN {X 0,Y 340.776,Z 398.036,A -85,B 0,C 180,E1 -14065.664,E2 -14065.664} C_VEL
LIN {X 0,Y 340.732,Z 398.039,A -85,B 0,C 180,E1 -14068.321,E2 -14068.321} C_VEL
LIN {X 0,Y 340.701,Z 398.048,A -85,B 0,C 180,E1 -14071.044,E2 -14071.044} C_VEL
LIN {X 0,Y 340.721,Z 398.044,A -85,B 0,C 180,E1 -14075.279,E2 -14075.279} C_VEL
LIN {X 0,Y 340.713,Z 398.044,A -85,B 0,C 180,E1 -14078.386,E2 -14078.386} C_VEL
LIN {X 0,Y 340.748,Z 398.17,A -85,B 0,C 180,E1 -14082.535,E2 -14082.535} C_VEL
LIN {X 0,Y 341.682,Z 403.184,A -85,B 0,C 180,E1 -14086.047,E2 -14086.047} C_VEL
LIN {X 0,Y 342.617,Z 408.296,A -85,B 0,C 180,E1 -14089.374,E2 -14089.374} C_VEL
LIN {X 0,Y 343.328,Z 412.759,A -85,B 0,C 180,E1 -14092.112,E2 -14092.112} C_VEL
LIN {X 0,Y 343.38,Z 416.594,A -85,B 0,C 180,E1 -14094.316,E2 -14094.316} C_VEL
LIN {X 0,Y 342.565,Z 422.956,A -85,B 0,C 180,E1 -14097.763,E2 -14097.763} C_VEL
LIN {X 0,Y 341.679,Z 430.549,A -85,B 0,C 180,E1 -14101.765,E2 -14101.765} C_VEL
LIN {X 0,Y 340.863,Z 438.03,A -85,B 0,C 180,E1 -14105.646,E2 -14105.646} C_VEL
LIN {X 0,Y 340.391,Z 443.766,A -85,B 0,C 180,E1 -14108.62,E2 -14108.62} C_VEL
LIN {X 0,Y 342.98,Z 457.807,A -85,B 0,C 180,E1 -14109.313,E2 -14109.313} C_VEL
LIN {X 0,Y 344.762,Z 471.402,A -85,B 0,C 180,E1 -14110.213,E2 -14110.213} C_VEL
LIN {X 0,Y 345.869,Z 482.924,A -85,B 0,C 180,E1 -14111.181,E2 -14111.181} C_VEL
LIN {X 0,Y 345.543,Z 489.353,A -85,B 0,C 180,E1 -14111.777,E2 -14111.777} C_VEL
LIN {X 0,Y 344.125,Z 501.183,A -85,B 0,C 180,E1 -14113.08,E2 -14113.08} C_VEL
LIN {X 0,Y 343.059,Z 510.302,A -85,B 0,C 180,E1 -14114.335,E2 -14114.335} C_VEL
LIN {X 0,Y 342.103,Z 518.643,A -85,B 0,C 180,E1 -14115.728,E2 -14115.728} C_VEL
LIN {X 0,Y 341.182,Z 525.988,A -85,B 0,C 180,E1 -14117.206,E2 -14117.206} C_VEL
LIN {X 0,Y 340.344,Z 533.231,A -85,B 0,C 180,E1 -14118.988,E2 -14118.988} C_VEL
LIN {X 0,Y 339.846,Z 538.128,A -85,B 0,C 180,E1 -14120.477,E2 -14120.477} C_VEL
LIN {X 0,Y 339.445,Z 542.894,A -85,B 0,C 180,E1 -14122.266,E2 -14122.266} C_VEL
LIN {X 0,Y 339.258,Z 546.543,A -85,B 0,C 180,E1 -14124.055,E2 -14124.055} C_VEL
LIN {X 0,Y 339.194,Z 548.427,A -85,B 0,C 180,E1 -14125.246,E2 -14125.246} C_VEL
LIN {X 0,Y 339.131,Z 549.84,A -85,B 0,C 180,E1 -14126.435,E2 -14126.435} C_VEL
LIN {X 0,Y 339.229,Z 551.473,A -85,B 0,C 180,E1 -14128.813,E2 -14128.813} C_VEL
LIN {X 0,Y 339.29,Z 551.695,A -85,B 0,C 180,E1 -14130,E2 -14130} C_VEL
LIN {X 0,Y 339.26,Z 551.473,A -85,B 0,C 180,E1 -14131.187,E2 -14131.187} C_VEL
LIN {X 0,Y 339.131,Z 549.837,A -85,B 0,C 180,E1 -14133.564,E2 -14133.564} C_VEL
LIN {X 0,Y 339.193,Z 548.422,A -85,B 0,C 180,E1 -14134.754,E2 -14134.754} C_VEL
LIN {X 0,Y 339.298,Z 545.449,A -85,B 0,C 180,E1 -14136.541,E2 -14136.541} C_VEL
LIN {X 0,Y 339.547,Z 541.429,A -85,B 0,C 180,E1 -14138.331,E2 -14138.331} C_VEL
LIN {X 0,Y 340.144,Z 535.263,A -85,B 0,C 180,E1 -14140.416,E2 -14140.416} C_VEL
LIN {X 0,Y 340.847,Z 528.532,A -85,B 0,C 180,E1 -14142.201,E2 -14142.201} C_VEL
LIN {X 0,Y 341.899,Z 520.2,A -85,B 0,C 180,E1 -14143.977,E2 -14143.977} C_VEL
LIN {X 0,Y 342.967,Z 511.665,A -85,B 0,C 180,E1 -14145.45,E2 -14145.45} C_VEL
LIN {X 0,Y 344.118,Z 501.122,A -85,B 0,C 180,E1 -14146.92,E2 -14146.92} C_VEL
LIN {X 0,Y 345.537,Z 489.281,A -85,B 0,C 180,E1 -14148.223,E2 -14148.223} C_VEL
LIN {X 0,Y 345.967,Z 484.55,A -85,B 0,C 180,E1 -14148.66,E2 -14148.66} C_VEL
LIN {X 0,Y 344.913,Z 472.627,A -85,B 0,C 180,E1 -14149.686,E2 -14149.686} C_VEL
LIN {X 0,Y 343.202,Z 459.298,A -85,B 0,C 180,E1 -14150.588,E2 -14150.588} C_VEL
LIN {X 0,Y 340.795,Z 446.064,A -85,B 0,C 180,E1 -14151.276,E2 -14151.276} C_VEL
LIN {X 0,Y 340.372,Z 443.686,A -85,B 0,C 180,E1 -14151.381,E2 -14151.381} C_VEL
LIN {X 0,Y 341.124,Z 435.523,A -85,B 0,C 180,E1 -14155.636,E2 -14155.636} C_VEL
LIN {X 0,Y 341.802,Z 429.26,A -85,B 0,C 180,E1 -14158.895,E2 -14158.895} C_VEL
LIN {X 0,Y 342.703,Z 421.886,A -85,B 0,C 180,E1 -14162.774,E2 -14162.774} C_VEL
LIN {X 0,Y 343.394,Z 416.482,A -85,B 0,C 180,E1 -14165.682,E2 -14165.682} C_VEL
LIN {X 0,Y 343.3,Z 412.635,A -85,B 0,C 180,E1 -14167.891,E2 -14167.891} C_VEL
LIN {X 0,Y 342.499,Z 407.523,A -85,B 0,C 180,E1 -14171.044,E2 -14171.044} C_VEL
LIN {X 0,Y 341.563,Z 402.478,A -85,B 0,C 180,E1 -14174.394,E2 -14174.394} C_VEL
LIN {X 0,Y 340.727,Z 398.047,A -85,B 0,C 180,E1 -14177.58,E2 -14177.58} C_VEL
LIN {X 0,Y 340.736,Z 398.04,A -85,B 0,C 180,E1 -14181.773,E2 -14181.773} C_VEL
LIN {X 0,Y 340.725,Z 398.041,A -85,B 0,C 180,E1 -14185.595,E2 -14185.595} C_VEL
LIN {X 0,Y 340.7,Z 398.048,A -85,B 0,C 180,E1 -14188.955,E2 -14188.955} C_VEL
LIN {X 0,Y 340.805,Z 398.033,A -85,B 0,C 180,E1 -14193.02,E2 -14193.02} C_VEL
LIN {X 0,Y 340.758,Z 398.036,A -85,B 0,C 180,E1 -14195.638,E2 -14195.638} C_VEL
LIN {X 0,Y 340.755,Z 398.036,A -85,B 0,C 180,E1 -14199.475,E2 -14199.475} C_VEL
LIN {X 0,Y 340.86,Z 398.024,A -85,B 0,C 180,E1 -14201.984,E2 -14201.984} C_VEL
LIN {X 0,Y 340.872,Z 398.022,A -85,B 0,C 180,E1 -14205.705,E2 -14205.705} C_VEL
LIN {X 0,Y 340.878,Z 398.021,A -85,B 0,C 180,E1 -14209.306,E2 -14209.306} C_VEL
LIN {X 0,Y 341.079,Z 397.998,A -85,B 0,C 180,E1 -14212.898,E2 -14212.898} C_VEL
LIN {X 0,Y 341.171,Z 397.985,A -85,B 0,C 180,E1 -14217.639,E2 -14217.639} C_VEL
LIN {X 0,Y 341.319,Z 397.968,A -85,B 0,C 180,E1 -14220,E2 -14220} C_VEL
LIN {X 0,Y 341.171,Z 397.99,A -85,B 0,C 180,E1 -14222.361,E2 -14222.361} C_VEL
LIN {X 0,Y 341.079,Z 397.995,A -85,B 0,C 180,E1 -14227.102,E2 -14227.102} C_VEL
LIN {X 0,Y 340.874,Z 398.023,A -85,B 0,C 180,E1 -14230.694,E2 -14230.694} C_VEL
LIN {X 0,Y 340.865,Z 398.026,A -85,B 0,C 180,E1 -14234.325,E2 -14234.325} C_VEL
LIN {X 0,Y 340.84,Z 398.027,A -85,B 0,C 180,E1 -14238.467,E2 -14238.467} C_VEL
LIN {X 0,Y 340.724,Z 398.044,A -85,B 0,C 180,E1 -14241.843,E2 -14241.843} C_VEL
LIN {X 0,Y 340.774,Z 398.036,A -85,B 0,C 180,E1 -14245.664,E2 -14245.664} C_VEL
LIN {X 0,Y 340.731,Z 398.041,A -85,B 0,C 180,E1 -14248.321,E2 -14248.321} C_VEL
LIN {X 0,Y 340.7,Z 398.043,A -85,B 0,C 180,E1 -14251.045,E2 -14251.045} C_VEL
LIN {X 0,Y 340.721,Z 398.041,A -85,B 0,C 180,E1 -14255.279,E2 -14255.279} C_VEL
LIN {X 0,Y 340.714,Z 398.042,A -85,B 0,C 180,E1 -14258.387,E2 -14258.387} C_VEL
LIN {X 0,Y 340.702,Z 398.045,A -85,B 0,C 180,E1 -14262.046,E2 -14262.046} C_VEL
LIN {X 0,Y 340.739,Z 398.042,A -85,B 0,C 180,E1 -14265.47,E2 -14265.47} C_VEL
LIN {X 0,Y 340.729,Z 398.04,A -85,B 0,C 180,E1 -14268.697,E2 -14268.697} C_VEL
LIN {X 0,Y 340.728,Z 398.044,A -85,B 0,C 180,E1 -14271.772,E2 -14271.772} C_VEL
LIN {X 0,Y 340.555,Z 398.063,A -85,B 0,C 180,E1 -14274.702,E2 -14274.702} C_VEL
LIN {X 0,Y 340.255,Z 398.103,A -85,B 0,C 180,E1 -14277.872,E2 -14277.872} C_VEL
LIN {X 0,Y 340.175,Z 398.566,A -85,B 0,C 180,E1 -14278.902,E2 -14278.902} C_VEL
LIN {X 0,Y 340.075,Z 401.992,A -85,B 0,C 180,E1 -14282.957,E2 -14282.957} C_VEL
LIN {X 0,Y 339.945,Z 405.548,A -85,B 0,C 180,E1 -14286.871,E2 -14286.871} C_VEL
LIN {X 0,Y 339.91,Z 407.32,A -85,B 0,C 180,E1 -14288.71,E2 -14288.71} C_VEL
LIN {X 0,Y 343.892,Z 420.625,A -85,B 0,C 180,E1 -14289.53,E2 -14289.53} C_VEL
LIN {X 0,Y 346.94,Z 432.941,A -85,B 0,C 180,E1 -14290.482,E2 -14290.482} C_VEL
LIN {X 0,Y 347.699,Z 436.872,A -85,B 0,C 180,E1 -14290.829,E2 -14290.829} C_VEL
LIN {X 0,Y 347.142,Z 445.622,A -85,B 0,C 180,E1 -14291.559,E2 -14291.559} C_VEL
LIN {X 0,Y 346.078,Z 456.26,A -85,B 0,C 180,E1 -14292.642,E2 -14292.642} C_VEL
LIN {X 0,Y 345.032,Z 466.069,A -85,B 0,C 180,E1 -14293.887,E2 -14293.887} C_VEL
LIN {X 0,Y 343.98,Z 474.576,A -85,B 0,C 180,E1 -14295.203,E2 -14295.203} C_VEL
LIN {X 0,Y 342.952,Z 482.407,A -85,B 0,C 180,E1 -14296.671,E2 -14296.671} C_VEL
LIN {X 0,Y 341.951,Z 490.054,A -85,B 0,C 180,E1 -14298.44,E2 -14298.44} C_VEL
LIN {X 0,Y 340.888,Z 497.075,A -85,B 0,C 180,E1 -14300.507,E2 -14300.507} C_VEL
LIN {X 0,Y 340.319,Z 502.056,A -85,B 0,C 180,E1 -14302.421,E2 -14302.421} C_VEL
LIN {X 0,Y 339.855,Z 505.313,A -85,B 0,C 180,E1 -14304.065,E2 -14304.065} C_VEL
LIN {X 0,Y 339.64,Z 507.157,A -85,B 0,C 180,E1 -14305.252,E2 -14305.252} C_VEL
LIN {X 0,Y 339.628,Z 508.535,A -85,B 0,C 180,E1 -14306.441,E2 -14306.441} C_VEL
LIN {X 0,Y 339.529,Z 509.521,A -85,B 0,C 180,E1 -14307.627,E2 -14307.627} C_VEL
LIN {X 0,Y 339.351,Z 510.363,A -85,B 0,C 180,E1 -14310,E2 -14310} C_VEL
LIN {X 0,Y 339.526,Z 509.587,A -85,B 0,C 180,E1 -14312.373,E2 -14312.373} C_VEL
LIN {X 0,Y 339.61,Z 508.629,A -85,B 0,C 180,E1 -14313.56,E2 -14313.56} C_VEL
LIN {X 0,Y 339.637,Z 507.29,A -85,B 0,C 180,E1 -14314.748,E2 -14314.748} C_VEL
LIN {X 0,Y 340.033,Z 504.44,A -85,B 0,C 180,E1 -14316.527,E2 -14316.527} C_VEL
LIN {X 0,Y 340.458,Z 500.582,A -85,B 0,C 180,E1 -14318.308,E2 -14318.308} C_VEL
LIN {X 0,Y 341.116,Z 495.597,A -85,B 0,C 180,E1 -14320.086,E2 -14320.086} C_VEL
LIN {X 0,Y 342.027,Z 489.311,A -85,B 0,C 180,E1 -14321.858,E2 -14321.858} C_VEL
LIN {X 0,Y 343.12,Z 481.441,A -85,B 0,C 180,E1 -14323.624,E2 -14323.624} C_VEL
LIN {X 0,Y 344.167,Z 473.414,A -85,B 0,C 180,E1 -14325.092,E2 -14325.092} C_VEL
LIN {X 0,Y 345.366,Z 463.611,A -85,B 0,C 180,E1 -14326.553,E2 -14326.553} C_VEL
LIN {X 0,Y 346.309,Z 453.965,A -85,B 0,C 180,E1 -14327.723,E2 -14327.723} C_VEL
LIN {X 0,Y 347.355,Z 443.502,A -85,B 0,C 180,E1 -14328.736,E2 -14328.736} C_VEL
LIN {X 0,Y 347.724,Z 436.582,A -85,B 0,C 180,E1 -14329.297,E2 -14329.297} C_VEL
LIN {X 0,Y 345.096,Z 425.027,A -85,B 0,C 180,E1 -14330.256,E2 -14330.256} C_VEL
LIN {X 0,Y 341.489,Z 412.441,A -85,B 0,C 180,E1 -14331.111,E2 -14331.111} C_VEL
LIN {X 0,Y 339.882,Z 407.252,A -85,B 0,C 180,E1 -14331.415,E2 -14331.415} C_VEL
LIN {X 0,Y 339.996,Z 404.303,A -85,B 0,C 180,E1 -14334.561,E2 -14334.561} C_VEL
LIN {X 0,Y 340.099,Z 400.946,A -85,B 0,C 180,E1 -14338.378,E2 -14338.378} C_VEL
LIN {X 0,Y 340.191,Z 398.663,A -85,B 0,C 180,E1 -14341.096,E2 -14341.096} C_VEL
LIN {X 0,Y 340.301,Z 398.098,A -85,B 0,C 180,E1 -14342.477,E2 -14342.477} C_VEL
LIN {X 0,Y 340.557,Z 398.062,A -85,B 0,C 180,E1 -14345.298,E2 -14345.298} C_VEL
LIN {X 0,Y 340.706,Z 398.047,A -85,B 0,C 180,E1 -14348.385,E2 -14348.385} C_VEL
LIN {X 0,Y 340.702,Z 398.045,A -85,B 0,C 180,E1 -14352.046,E2 -14352.046} C_VEL
LIN {X 0,Y 340.655,Z 398.053,A -85,B 0,C 180,E1 -14356.227,E2 -14356.227} C_VEL
LIN {X 0,Y 340.681,Z 398.045,A -85,B 0,C 180,E1 -14357.513,E2 -14357.513} C_VEL
LIN {X 0,Y 340.035,Z 398.13,A -85,B 0,C 180,E1 -14358.501,E2 -14358.501} C_VEL
LIN {X 0,Y 337.184,Z 398.489,A -85,B 0,C 180,E1 -14360.107,E2 -14360.107} C_VEL
LIN {X 0,Y 334.761,Z 398.79,A -85,B 0,C 180,E1 -14361.408,E2 -14361.408} C_VEL
LIN {X 0,Y 333.733,Z 398.915,A -85,B 0,C 180,E1 -14362.415,E2 -14362.415} C_VEL
LIN {X 0,Y 333.656,Z 398.922,A -85,B 0,C 180,E1 -14362.756,E2 -14362.756} C_VEL
LIN {X 0,Y 333.678,Z 398.917,A -85,B 0,C 180,E1 -14365.342,E2 -14365.342} C_VEL
LIN {X 0,Y 333.694,Z 398.917,A -85,B 0,C 180,E1 -14369.637,E2 -14369.637} C_VEL
LIN {X 0,Y 333.743,Z 398.913,A -85,B 0,C 180,E1 -14372.401,E2 -14372.401} C_VEL
LIN {X 0,Y 333.729,Z 398.911,A -85,B 0,C 180,E1 -14375.091,E2 -14375.091} C_VEL
LIN {X 0,Y 333.677,Z 398.918,A -85,B 0,C 180,E1 -14379.019,E2 -14379.019} C_VEL
LIN {X 0,Y 333.798,Z 398.905,A -85,B 0,C 180,E1 -14381.59,E2 -14381.59} C_VEL
LIN {X 0,Y 333.812,Z 398.904,A -85,B 0,C 180,E1 -14385.577,E2 -14385.577} C_VEL
LIN {X 0,Y 333.837,Z 398.898,A -85,B 0,C 180,E1 -14389.078,E2 -14389.078} C_VEL
LIN {X 0,Y 333.998,Z 398.878,A -85,B 0,C 180,E1 -14392.747,E2 -14392.747} C_VEL
LIN {X 0,Y 333.811,Z 398.902,A -85,B 0,C 180,E1 -14395.169,E2 -14395.169} C_VEL
LIN {X 0,Y 334.109,Z 398.869,A -85,B 0,C 180,E1 -14397.589,E2 -14397.589} C_VEL
LIN {X 0,Y 334.25,Z 398.85,A -85,B 0,C 180,E1 -14400,E2 -14400} C_VEL
LIN {X 0,Y 334.11,Z 398.865,A -85,B 0,C 180,E1 -14402.411,E2 -14402.411} C_VEL
LIN {X 0,Y 334.03,Z 398.877,A -85,B 0,C 180,E1 -14407.252,E2 -14407.252} C_VEL
LIN {X 0,Y 333.842,Z 398.899,A -85,B 0,C 180,E1 -14410.922,E2 -14410.922} C_VEL
LIN {X 0,Y 333.812,Z 398.901,A -85,B 0,C 180,E1 -14414.634,E2 -14414.634} C_VEL
LIN {X 0,Y 333.8,Z 398.902,A -85,B 0,C 180,E1 -14418.655,E2 -14418.655} C_VEL
LIN {X 0,Y 333.696,Z 398.915,A -85,B 0,C 180,E1 -14422.278,E2 -14422.278} C_VEL
LIN {X 0,Y 333.738,Z 398.911,A -85,B 0,C 180,E1 -14426.246,E2 -14426.246} C_VEL
LIN {X 0,Y 333.693,Z 398.919,A -85,B 0,C 180,E1 -14428.974,E2 -14428.974} C_VEL
LIN {X 0,Y 333.646,Z 398.923,A -85,B 0,C 180,E1 -14432.587,E2 -14432.587} C_VEL
LIN {X 0,Y 333.679,Z 398.919,A -85,B 0,C 180,E1 -14436.139,E2 -14436.139} C_VEL
LIN {X 0,Y 333.65,Z 398.926,A -85,B 0,C 180,E1 -14439.192,E2 -14439.192} C_VEL
LIN {X 0,Y 333.695,Z 398.967,A -85,B 0,C 180,E1 -14441.966,E2 -14441.966} C_VEL
LIN {X 0,Y 334.62,Z 403.94,A -85,B 0,C 180,E1 -14445.57,E2 -14445.57} C_VEL
LIN {X 0,Y 335.687,Z 409.864,A -85,B 0,C 180,E1 -14449.532,E2 -14449.532} C_VEL
LIN {X 0,Y 336.421,Z 414.993,A -85,B 0,C 180,E1 -14452.711,E2 -14452.711} C_VEL
LIN {X 0,Y 336.293,Z 418.222,A -85,B 0,C 180,E1 -14454.591,E2 -14454.591} C_VEL
LIN {X 0,Y 335.532,Z 423.867,A -85,B 0,C 180,E1 -14457.715,E2 -14457.715} C_VEL
LIN {X 0,Y 334.562,Z 431.65,A -85,B 0,C 180,E1 -14461.918,E2 -14461.918} C_VEL
LIN {X 0,Y 333.772,Z 438.849,A -85,B 0,C 180,E1 -14465.757,E2 -14465.757} C_VEL
LIN {X 0,Y 333.378,Z 443.338,A -85,B 0,C 180,E1 -14468.148,E2 -14468.148} C_VEL
LIN {X 0,Y 335.953,Z 456.992,A -85,B 0,C 180,E1 -14468.841,E2 -14468.841} C_VEL
LIN {X 0,Y 337.679,Z 469.752,A -85,B 0,C 180,E1 -14469.697,E2 -14469.697} C_VEL
LIN {X 0,Y 338.888,Z 482.48,A -85,B 0,C 180,E1 -14470.778,E2 -14470.778} C_VEL
LIN {X 0,Y 338.944,Z 487.383,A -85,B 0,C 180,E1 -14471.253,E2 -14471.253} C_VEL
LIN {X 0,Y 337.627,Z 498.391,A -85,B 0,C 180,E1 -14472.432,E2 -14472.432} C_VEL
LIN {X 0,Y 336.359,Z 508.435,A -85,B 0,C 180,E1 -14473.788,E2 -14473.788} C_VEL
LIN {X 0,Y 335.2,Z 518.211,A -85,B 0,C 180,E1 -14475.428,E2 -14475.428} C_VEL
LIN {X 0,Y 334.232,Z 525.555,A -85,B 0,C 180,E1 -14476.936,E2 -14476.936} C_VEL
LIN {X 0,Y 333.321,Z 532.797,A -85,B 0,C 180,E1 -14478.753,E2 -14478.753} C_VEL
LIN {X 0,Y 332.82,Z 537.695,A -85,B 0,C 180,E1 -14480.274,E2 -14480.274} C_VEL
LIN {X 0,Y 332.39,Z 542.461,A -85,B 0,C 180,E1 -14482.1,E2 -14482.1} C_VEL
LIN {X 0,Y 332.181,Z 546.11,A -85,B 0,C 180,E1 -14483.927,E2 -14483.927} C_VEL
LIN {X 0,Y 332.116,Z 547.995,A -85,B 0,C 180,E1 -14485.144,E2 -14485.144} C_VEL
LIN {X 0,Y 332.058,Z 549.409,A -85,B 0,C 180,E1 -14486.359,E2 -14486.359} C_VEL
LIN {X 0,Y 332.136,Z 551.041,A -85,B 0,C 180,E1 -14488.787,E2 -14488.787} C_VEL
LIN {X 0,Y 332.213,Z 551.264,A -85,B 0,C 180,E1 -14490,E2 -14490} C_VEL
LIN {X 0,Y 332.166,Z 551.04,A -85,B 0,C 180,E1 -14491.212,E2 -14491.212} C_VEL
LIN {X 0,Y 332.058,Z 549.405,A -85,B 0,C 180,E1 -14493.64,E2 -14493.64} C_VEL
LIN {X 0,Y 332.115,Z 547.989,A -85,B 0,C 180,E1 -14494.856,E2 -14494.856} C_VEL
LIN {X 0,Y 332.219,Z 545.013,A -85,B 0,C 180,E1 -14496.681,E2 -14496.681} C_VEL
LIN {X 0,Y 332.493,Z 540.993,A -85,B 0,C 180,E1 -14498.509,E2 -14498.509} C_VEL
LIN {X 0,Y 333.129,Z 534.827,A -85,B 0,C 180,E1 -14500.638,E2 -14500.638} C_VEL
LIN {X 0,Y 333.888,Z 528.097,A -85,B 0,C 180,E1 -14502.46,E2 -14502.46} C_VEL
LIN {X 0,Y 334.962,Z 519.762,A -85,B 0,C 180,E1 -14504.272,E2 -14504.272} C_VEL
LIN {X 0,Y 336.092,Z 510.652,A -85,B 0,C 180,E1 -14505.865,E2 -14505.865} C_VEL
LIN {X 0,Y 337.328,Z 500.686,A -85,B 0,C 180,E1 -14507.271,E2 -14507.271} C_VEL
LIN {X 0,Y 338.784,Z 488.843,A -85,B 0,C 180,E1 -14508.599,E2 -14508.599} C_VEL
LIN {X 0,Y 338.993,Z 484.096,A -85,B 0,C 180,E1 -14509.058,E2 -14509.058} C_VEL
LIN {X 0,Y 337.927,Z 471.7,A -85,B 0,C 180,E1 -14510.142,E2 -14510.142} C_VEL
LIN {X 0,Y 336.158,Z 458.231,A -85,B 0,C 180,E1 -14511.071,E2 -14511.071} C_VEL
LIN {X 0,Y 333.659,Z 445.085,A -85,B 0,C 180,E1 -14511.769,E2 -14511.769} C_VEL
LIN {X 0,Y 333.377,Z 443.264,A -85,B 0,C 180,E1 -14511.853,E2 -14511.853} C_VEL
LIN {X 0,Y 333.981,Z 437.035,A -85,B 0,C 180,E1 -14515.196,E2 -14515.196} C_VEL
LIN {X 0,Y 334.731,Z 430.144,A -85,B 0,C 180,E1 -14518.876,E2 -14518.876} C_VEL
LIN {X 0,Y 335.543,Z 423.843,A -85,B 0,C 180,E1 -14522.283,E2 -14522.283} C_VEL
LIN {X 0,Y 336.415,Z 417.453,A -85,B 0,C 180,E1 -14525.799,E2 -14525.799} C_VEL
LIN {X 0,Y 336.291,Z 413.584,A -85,B 0,C 180,E1 -14528.08,E2 -14528.08} C_VEL
LIN {X 0,Y 335.542,Z 408.851,A -85,B 0,C 180,E1 -14531.059,E2 -14531.059} C_VEL
LIN {X 0,Y 334.614,Z 403.86,A -85,B 0,C 180,E1 -14534.429,E2 -14534.429} C_VEL
LIN {X 0,Y 333.67,Z 398.927,A -85,B 0,C 180,E1 -14538.131,E2 -14538.131} C_VEL
LIN {X 0,Y 333.655,Z 398.923,A -85,B 0,C 180,E1 -14542.349,E2 -14542.349} C_VEL
LIN {X 0,Y 333.676,Z 398.921,A -85,B 0,C 180,E1 -14545.341,E2 -14545.341} C_VEL
LIN {X 0,Y 333.692,Z 398.916,A -85,B 0,C 180,E1 -14549.637,E2 -14549.637} C_VEL
LIN {X 0,Y 333.742,Z 398.913,A -85,B 0,C 180,E1 -14552.401,E2 -14552.401} C_VEL
LIN {X 0,Y 333.729,Z 398.914,A -85,B 0,C 180,E1 -14555.091,E2 -14555.091} C_VEL
LIN {X 0,Y 333.687,Z 398.919,A -85,B 0,C 180,E1 -14559.02,E2 -14559.02} C_VEL
LIN {X 0,Y 333.796,Z 398.903,A -85,B 0,C 180,E1 -14561.59,E2 -14561.59} C_VEL
LIN {X 0,Y 333.811,Z 398.901,A -85,B 0,C 180,E1 -14565.577,E2 -14565.577} C_VEL
LIN {X 0,Y 333.841,Z 398.899,A -85,B 0,C 180,E1 -14569.078,E2 -14569.078} C_VEL
LIN {X 0,Y 334.029,Z 398.877,A -85,B 0,C 180,E1 -14572.748,E2 -14572.748} C_VEL
LIN {X 0,Y 333.813,Z 398.901,A -85,B 0,C 180,E1 -14575.169,E2 -14575.169} C_VEL
LIN {X 0,Y 334.108,Z 398.864,A -85,B 0,C 180,E1 -14577.589,E2 -14577.589} C_VEL
LIN {X 0,Y 334.269,Z 398.846,A -85,B 0,C 180,E1 -14580,E2 -14580} C_VEL
LIN {X 0,Y 334.108,Z 398.869,A -85,B 0,C 180,E1 -14582.411,E2 -14582.411} C_VEL
LIN {X 0,Y 334.029,Z 398.873,A -85,B 0,C 180,E1 -14587.252,E2 -14587.252} C_VEL
LIN {X 0,Y 333.837,Z 398.898,A -85,B 0,C 180,E1 -14590.922,E2 -14590.922} C_VEL
LIN {X 0,Y 333.811,Z 398.902,A -85,B 0,C 180,E1 -14594.634,E2 -14594.634} C_VEL
LIN {X 0,Y 333.799,Z 398.903,A -85,B 0,C 180,E1 -14598.655,E2 -14598.655} C_VEL
LIN {X 0,Y 333.663,Z 398.923,A -85,B 0,C 180,E1 -14602.28,E2 -14602.28} C_VEL
LIN {X 0,Y 333.737,Z 398.913,A -85,B 0,C 180,E1 -14606.246,E2 -14606.246} C_VEL
LIN {X 0,Y 333.692,Z 398.916,A -85,B 0,C 180,E1 -14608.974,E2 -14608.974} C_VEL
LIN {X 0,Y 333.648,Z 398.92,A -85,B 0,C 180,E1 -14612.588,E2 -14612.588} C_VEL
LIN {X 0,Y 333.68,Z 398.919,A -85,B 0,C 180,E1 -14616.139,E2 -14616.139} C_VEL
LIN {X 0,Y 333.65,Z 398.922,A -85,B 0,C 180,E1 -14619.192,E2 -14619.192} C_VEL
LIN {X 0,Y 333.636,Z 398.923,A -85,B 0,C 180,E1 -14622.5,E2 -14622.5} C_VEL
LIN {X 0,Y 333.677,Z 398.921,A -85,B 0,C 180,E1 -14625.968,E2 -14625.968} C_VEL
LIN {X 0,Y 333.704,Z 398.918,A -85,B 0,C 180,E1 -14629.304,E2 -14629.304} C_VEL
LIN {X 0,Y 333.634,Z 398.927,A -85,B 0,C 180,E1 -14633.175,E2 -14633.175} C_VEL
LIN {X 0,Y 333.301,Z 398.972,A -85,B 0,C 180,E1 -14636.754,E2 -14636.754} C_VEL
LIN {X 0,Y 333.159,Z 398.987,A -85,B 0,C 180,E1 -14638.172,E2 -14638.172} C_VEL
LIN {X 0,Y 333.075,Z 401.239,A -85,B 0,C 180,E1 -14640.967,E2 -14640.967} C_VEL
LIN {X 0,Y 332.978,Z 403.567,A -85,B 0,C 180,E1 -14643.689,E2 -14643.689} C_VEL
LIN {X 0,Y 332.906,Z 405.976,A -85,B 0,C 180,E1 -14646.352,E2 -14646.352} C_VEL
LIN {X 0,Y 332.848,Z 407.746,A -85,B 0,C 180,E1 -14648.222,E2 -14648.222} C_VEL
LIN {X 0,Y 337.217,Z 422.041,A -85,B 0,C 180,E1 -14649.157,E2 -14649.157} C_VEL
LIN {X 0,Y 340.147,Z 434.015,A -85,B 0,C 180,E1 -14650.121,E2 -14650.121} C_VEL
LIN {X 0,Y 341.042,Z 439.367,A -85,B 0,C 180,E1 -14650.605,E2 -14650.605} C_VEL
LIN {X 0,Y 339.966,Z 450.632,A -85,B 0,C 180,E1 -14651.624,E2 -14651.624} C_VEL
LIN {X 0,Y 338.867,Z 461.702,A -85,B 0,C 180,E1 -14652.905,E2 -14652.905} C_VEL
LIN {X 0,Y 337.639,Z 471.441,A -85,B 0,C 180,E1 -14654.3,E2 -14654.3} C_VEL
LIN {X 0,Y 336.47,Z 479.898,A -85,B 0,C 180,E1 -14655.793,E2 -14655.793} C_VEL
LIN {X 0,Y 335.295,Z 488.109,A -85,B 0,C 180,E1 -14657.594,E2 -14657.594} C_VEL
LIN {X 0,Y 334.478,Z 493.723,A -85,B 0,C 180,E1 -14659.099,E2 -14659.099} C_VEL
LIN {X 0,Y 333.692,Z 499.19,A -85,B 0,C 180,E1 -14660.912,E2 -14660.912} C_VEL
LIN {X 0,Y 333.13,Z 503.477,A -85,B 0,C 180,E1 -14662.728,E2 -14662.728} C_VEL
LIN {X 0,Y 332.828,Z 505.744,A -85,B 0,C 180,E1 -14663.939,E2 -14663.939} C_VEL
LIN {X 0,Y 332.578,Z 507.589,A -85,B 0,C 180,E1 -14665.151,E2 -14665.151} C_VEL
LIN {X 0,Y 332.544,Z 508.968,A -85,B 0,C 180,E1 -14666.365,E2 -14666.365} C_VEL
LIN {X 0,Y 332.456,Z 509.952,A -85,B 0,C 180,E1 -14667.577,E2 -14667.577} C_VEL
LIN {X 0,Y 332.29,Z 510.793,A -85,B 0,C 180,E1 -14670,E2 -14670} C_VEL
LIN {X 0,Y 332.453,Z 510.018,A -85,B 0,C 180,E1 -14672.423,E2 -14672.423} C_VEL
LIN {X 0,Y 332.527,Z 509.06,A -85,B 0,C 180,E1 -14673.635,E2 -14673.635} C_VEL
LIN {X 0,Y 332.575,Z 507.721,A -85,B 0,C 180,E1 -14674.849,E2 -14674.849} C_VEL
LIN {X 0,Y 333.007,Z 504.87,A -85,B 0,C 180,E1 -14676.666,E2 -14676.666} C_VEL
LIN {X 0,Y 333.448,Z 501.012,A -85,B 0,C 180,E1 -14678.484,E2 -14678.484} C_VEL
LIN {X 0,Y 334.145,Z 496.027,A -85,B 0,C 180,E1 -14680.299,E2 -14680.299} C_VEL
LIN {X 0,Y 335.088,Z 489.741,A -85,B 0,C 180,E1 -14682.107,E2 -14682.107} C_VEL
LIN {X 0,Y 336.246,Z 481.869,A -85,B 0,C 180,E1 -14683.908,E2 -14683.908} C_VEL
LIN {X 0,Y 337.321,Z 473.843,A -85,B 0,C 180,E1 -14685.405,E2 -14685.405} C_VEL
LIN {X 0,Y 338.586,Z 464.038,A -85,B 0,C 180,E1 -14686.894,E2 -14686.894} C_VEL
LIN {X 0,Y 339.572,Z 454.391,A -85,B 0,C 180,E1 -14688.087,E2 -14688.087} C_VEL
LIN {X 0,Y 340.671,Z 443.926,A -85,B 0,C 180,E1 -14689.117,E2 -14689.117} C_VEL
LIN {X 0,Y 341.061,Z 438.401,A -85,B 0,C 180,E1 -14689.578,E2 -14689.578} C_VEL
LIN {X 0,Y 338.595,Z 427.285,A -85,B 0,C 180,E1 -14690.549,E2 -14690.549} C_VEL
LIN {X 0,Y 335.071,Z 414.837,A -85,B 0,C 180,E1 -14691.449,E2 -14691.449} C_VEL
LIN {X 0,Y 332.832,Z 407.692,A -85,B 0,C 180,E1 -14691.886,E2 -14691.886} C_VEL
LIN {X 0,Y 332.936,Z 404.849,A -85,B 0,C 180,E1 -14694.973,E2 -14694.973} C_VEL
LIN {X 0,Y 333.094,Z 401.342,A -85,B 0,C 180,E1 -14699.031,E2 -14699.031} C_VEL
LIN {X 0,Y 333.176,Z 399.041,A -85,B 0,C 180,E1 -14701.827,E2 -14701.827} C_VEL
LIN {X 0,Y 333.471,Z 398.949,A -85,B 0,C 180,E1 -14704.72,E2 -14704.72} C_VEL
LIN {X 0,Y 333.638,Z 398.923,A -85,B 0,C 180,E1 -14707.653,E2 -14707.653} C_VEL
LIN {X 0,Y 333.65,Z 398.924,A -85,B 0,C 180,E1 -14710.767,E2 -14710.767} C_VEL
LIN {X 0,Y 333.596,Z 398.932,A -85,B 0,C 180,E1 -14714.251,E2 -14714.251} C_VEL
LIN {X 0,Y 333.645,Z 398.922,A -85,B 0,C 180,E1 -14717.619,E2 -14717.619} C_VEL
LIN {X 0,Y 333.657,Z 398.919,A -85,B 0,C 180,E1 -14721.202,E2 -14721.202} C_VEL
LIN {X 0,Y 333.656,Z 398.922,A -85,B 0,C 180,E1 -14722.756,E2 -14722.756} C_VEL
LIN {X 0,Y 333.005,Z 399.005,A -85,B 0,C 180,E1 -14723.763,E2 -14723.763} C_VEL
LIN {X 0,Y 330.151,Z 399.356,A -85,B 0,C 180,E1 -14725.403,E2 -14725.403} C_VEL
LIN {X 0,Y 327.718,Z 399.661,A -85,B 0,C 180,E1 -14726.731,E2 -14726.731} C_VEL
LIN {X 0,Y 326.667,Z 399.793,A -85,B 0,C 180,E1 -14727.759,E2 -14727.759} C_VEL
LIN {X 0,Y 326.579,Z 399.799,A -85,B 0,C 180,E1 -14728.107,E2 -14728.107} C_VEL
LIN {X 0,Y 326.66,Z 399.796,A -85,B 0,C 180,E1 -14731.898,E2 -14731.898} C_VEL
LIN {X 0,Y 326.691,Z 399.789,A -85,B 0,C 180,E1 -14734.627,E2 -14734.627} C_VEL
LIN {X 0,Y 326.623,Z 399.798,A -85,B 0,C 180,E1 -14738.544,E2 -14738.544} C_VEL
LIN {X 0,Y 326.748,Z 399.781,A -85,B 0,C 180,E1 -14741.178,E2 -14741.178} C_VEL
LIN {X 0,Y 326.767,Z 399.78,A -85,B 0,C 180,E1 -14745.433,E2 -14745.433} C_VEL
LIN {X 0,Y 326.774,Z 399.778,A -85,B 0,C 180,E1 -14748.839,E2 -14748.839} C_VEL
LIN {X 0,Y 326.947,Z 399.756,A -85,B 0,C 180,E1 -14752.59,E2 -14752.59} C_VEL
LIN {X 0,Y 326.988,Z 399.757,A -85,B 0,C 180,E1 -14753.831,E2 -14753.831} C_VEL
LIN {X 0,Y 327.05,Z 399.748,A -85,B 0,C 180,E1 -14757.537,E2 -14757.537} C_VEL
LIN {X 0,Y 327.202,Z 399.728,A -85,B 0,C 180,E1 -14760,E2 -14760} C_VEL
LIN {X 0,Y 327.05,Z 399.745,A -85,B 0,C 180,E1 -14762.463,E2 -14762.463} C_VEL
LIN {X 0,Y 327.001,Z 399.751,A -85,B 0,C 180,E1 -14766.169,E2 -14766.169} C_VEL
LIN {X 0,Y 326.919,Z 399.76,A -85,B 0,C 180,E1 -14768.655,E2 -14768.655} C_VEL
LIN {X 0,Y 326.743,Z 399.782,A -85,B 0,C 180,E1 -14772.421,E2 -14772.421} C_VEL
LIN {X 0,Y 326.758,Z 399.781,A -85,B 0,C 180,E1 -14774.957,E2 -14774.957} C_VEL
LIN {X 0,Y 326.736,Z 399.783,A -85,B 0,C 180,E1 -14778.838,E2 -14778.838} C_VEL
LIN {X 0,Y 326.624,Z 399.798,A -85,B 0,C 180,E1 -14782.787,E2 -14782.787} C_VEL
LIN {X 0,Y 326.693,Z 399.792,A -85,B 0,C 180,E1 -14785.484,E2 -14785.484} C_VEL
LIN {X 0,Y 326.651,Z 399.796,A -85,B 0,C 180,E1 -14789.66,E2 -14789.66} C_VEL
LIN {X 0,Y 326.61,Z 399.799,A -85,B 0,C 180,E1 -14794.019,E2 -14794.019} C_VEL
LIN {X 0,Y 326.631,Z 399.799,A -85,B 0,C 180,E1 -14797.238,E2 -14797.238} C_VEL
LIN {X 0,Y 326.636,Z 399.8,A -85,B 0,C 180,E1 -14801.382,E2 -14801.382} C_VEL
LIN {X 0,Y 327.521,Z 404.707,A -85,B 0,C 180,E1 -14805.082,E2 -14805.082} C_VEL
LIN {X 0,Y 328.436,Z 409.63,A -85,B 0,C 180,E1 -14808.499,E2 -14808.499} C_VEL
LIN {X 0,Y 329.365,Z 415.26,A -85,B 0,C 180,E1 -14812.14,E2 -14812.14} C_VEL
LIN {X 0,Y 329.346,Z 418.66,A -85,B 0,C 180,E1 -14814.183,E2 -14814.183} C_VEL
LIN {X 0,Y 328.49,Z 424.777,A -85,B 0,C 180,E1 -14817.664,E2 -14817.664} C_VEL
LIN {X 0,Y 327.581,Z 431.852,A -85,B 0,C 180,E1 -14821.597,E2 -14821.597} C_VEL
LIN {X 0,Y 326.809,Z 438.432,A -85,B 0,C 180,E1 -14825.206,E2 -14825.206} C_VEL
LIN {X 0,Y 326.38,Z 442.975,A -85,B 0,C 180,E1 -14827.661,E2 -14827.661} C_VEL
LIN {X 0,Y 328.971,Z 456.466,A -85,B 0,C 180,E1 -14828.365,E2 -14828.365} C_VEL
LIN {X 0,Y 330.736,Z 468.947,A -85,B 0,C 180,E1 -14829.225,E2 -14829.225} C_VEL
LIN {X 0,Y 331.919,Z 482.035,A -85,B 0,C 180,E1 -14830.358,E2 -14830.358} C_VEL
LIN {X 0,Y 332.181,Z 486.952,A -85,B 0,C 180,E1 -14830.856,E2 -14830.856} C_VEL
LIN {X 0,Y 330.854,Z 497.962,A -85,B 0,C 180,E1 -14832.06,E2 -14832.06} C_VEL
LIN {X 0,Y 329.647,Z 506.918,A -85,B 0,C 180,E1 -14833.272,E2 -14833.272} C_VEL
LIN {X 0,Y 328.535,Z 516.358,A -85,B 0,C 180,E1 -14834.85,E2 -14834.85} C_VEL
LIN {X 0,Y 327.295,Z 525.123,A -85,B 0,C 180,E1 -14836.654,E2 -14836.654} C_VEL
LIN {X 0,Y 326.296,Z 532.362,A -85,B 0,C 180,E1 -14838.508,E2 -14838.508} C_VEL
LIN {X 0,Y 325.803,Z 537.263,A -85,B 0,C 180,E1 -14840.062,E2 -14840.062} C_VEL
LIN {X 0,Y 325.333,Z 542.028,A -85,B 0,C 180,E1 -14841.928,E2 -14841.928} C_VEL
LIN {X 0,Y 325.103,Z 545.939,A -85,B 0,C 180,E1 -14843.945,E2 -14843.945} C_VEL
LIN {X 0,Y 324.986,Z 548.977,A -85,B 0,C 180,E1 -14846.28,E2 -14846.28} C_VEL
LIN {X 0,Y 325.043,Z 550.609,A -85,B 0,C 180,E1 -14848.761,E2 -14848.761} C_VEL
LIN {X 0,Y 325.138,Z 550.833,A -85,B 0,C 180,E1 -14850,E2 -14850} C_VEL
LIN {X 0,Y 325.071,Z 550.608,A -85,B 0,C 180,E1 -14851.239,E2 -14851.239} C_VEL
LIN {X 0,Y 324.986,Z 548.973,A -85,B 0,C 180,E1 -14853.72,E2 -14853.72} C_VEL
LIN {X 0,Y 325.083,Z 545.984,A -85,B 0,C 180,E1 -14856.022,E2 -14856.022} C_VEL
LIN {X 0,Y 325.301,Z 542.005,A -85,B 0,C 180,E1 -14858.073,E2 -14858.073} C_VEL
LIN {X 0,Y 325.802,Z 537.236,A -85,B 0,C 180,E1 -14859.937,E2 -14859.937} C_VEL
LIN {X 0,Y 326.562,Z 530.075,A -85,B 0,C 180,E1 -14862.112,E2 -14862.112} C_VEL
LIN {X 0,Y 327.711,Z 522.327,A -85,B 0,C 180,E1 -14863.961,E2 -14863.961} C_VEL
LIN {X 0,Y 328.984,Z 512.602,A -85,B 0,C 180,E1 -14865.805,E2 -14865.805} C_VEL
LIN {X 0,Y 330.178,Z 502.571,A -85,B 0,C 180,E1 -14867.337,E2 -14867.337} C_VEL
LIN {X 0,Y 331.657,Z 491.268,A -85,B 0,C 180,E1 -14868.694,E2 -14868.694} C_VEL
LIN {X 0,Y 332.147,Z 485.251,A -85,B 0,C 180,E1 -14869.306,E2 -14869.306} C_VEL
LIN {X 0,Y 331.272,Z 473.789,A -85,B 0,C 180,E1 -14870.374,E2 -14870.374} C_VEL
LIN {X 0,Y 329.642,Z 460.724,A -85,B 0,C 180,E1 -14871.351,E2 -14871.351} C_VEL
LIN {X 0,Y 327.387,Z 447.942,A -85,B 0,C 180,E1 -14872.092,E2 -14872.092} C_VEL
LIN {X 0,Y 326.393,Z 442.858,A -85,B 0,C 180,E1 -14872.33,E2 -14872.33} C_VEL
LIN {X 0,Y 327.074,Z 435.962,A -85,B 0,C 180,E1 -14876.135,E2 -14876.135} C_VEL
LIN {X 0,Y 327.824,Z 429.76,A -85,B 0,C 180,E1 -14879.543,E2 -14879.543} C_VEL
LIN {X 0,Y 328.665,Z 423.679,A -85,B 0,C 180,E1 -14882.932,E2 -14882.932} C_VEL
LIN {X 0,Y 329.382,Z 418.538,A -85,B 0,C 180,E1 -14885.825,E2 -14885.825} C_VEL
LIN {X 0,Y 329.352,Z 415.15,A -85,B 0,C 180,E1 -14887.858,E2 -14887.858} C_VEL
LIN {X 0,Y 328.418,Z 409.445,A -85,B 0,C 180,E1 -14891.559,E2 -14891.559} C_VEL
LIN {X 0,Y 327.471,Z 404.371,A -85,B 0,C 180,E1 -14895.091,E2 -14895.091} C_VEL
LIN {X 0,Y 326.612,Z 399.808,A -85,B 0,C 180,E1 -14898.564,E2 -14898.564} C_VEL
LIN {X 0,Y 326.626,Z 399.8,A -85,B 0,C 180,E1 -14901.392,E2 -14901.392} C_VEL
LIN {X 0,Y 326.622,Z 399.802,A -85,B 0,C 180,E1 -14904.851,E2 -14904.851} C_VEL
LIN {X 0,Y 326.612,Z 399.8,A -85,B 0,C 180,E1 -14907.456,E2 -14907.456} C_VEL
LIN {X 0,Y 326.65,Z 399.796,A -85,B 0,C 180,E1 -14910.34,E2 -14910.34} C_VEL
LIN {X 0,Y 326.692,Z 399.792,A -85,B 0,C 180,E1 -14914.516,E2 -14914.516} C_VEL
LIN {X 0,Y 326.651,Z 399.798,A -85,B 0,C 180,E1 -14918.546,E2 -14918.546} C_VEL
LIN {X 0,Y 326.747,Z 399.783,A -85,B 0,C 180,E1 -14921.178,E2 -14921.178} C_VEL
LIN {X 0,Y 326.766,Z 399.779,A -85,B 0,C 180,E1 -14925.433,E2 -14925.433} C_VEL
LIN {X 0,Y 326.776,Z 399.78,A -85,B 0,C 180,E1 -14928.839,E2 -14928.839} C_VEL
LIN {X 0,Y 326.983,Z 399.757,A -85,B 0,C 180,E1 -14932.59,E2 -14932.59} C_VEL
LIN {X 0,Y 326.78,Z 399.778,A -85,B 0,C 180,E1 -14935.065,E2 -14935.065} C_VEL
LIN {X 0,Y 327.049,Z 399.744,A -85,B 0,C 180,E1 -14937.537,E2 -14937.537} C_VEL
LIN {X 0,Y 327.22,Z 399.724,A -85,B 0,C 180,E1 -14940,E2 -14940} C_VEL
LIN {X 0,Y 327.049,Z 399.748,A -85,B 0,C 180,E1 -14942.463,E2 -14942.463} C_VEL
LIN {X 0,Y 326.974,Z 399.753,A -85,B 0,C 180,E1 -14946.676,E2 -14946.676} C_VEL
LIN {X 0,Y 326.817,Z 399.775,A -85,B 0,C 180,E1 -14949.906,E2 -14949.906} C_VEL
LIN {X 0,Y 326.762,Z 399.78,A -85,B 0,C 180,E1 -14953.685,E2 -14953.685} C_VEL
LIN {X 0,Y 326.702,Z 399.788,A -85,B 0,C 180,E1 -14957.528,E2 -14957.528} C_VEL
LIN {X 0,Y 326.662,Z 399.797,A -85,B 0,C 180,E1 -14960.135,E2 -14960.135} C_VEL
LIN {X 0,Y 326.652,Z 399.797,A -85,B 0,C 180,E1 -14964.129,E2 -14964.129} C_VEL
LIN {X 0,Y 326.685,Z 399.788,A -85,B 0,C 180,E1 -14966.858,E2 -14966.858} C_VEL
LIN {X 0,Y 326.636,Z 399.795,A -85,B 0,C 180,E1 -14970.61,E2 -14970.61} C_VEL
LIN {X 0,Y 326.61,Z 399.802,A -85,B 0,C 180,E1 -14974.019,E2 -14974.019} C_VEL
LIN {X 0,Y 326.632,Z 399.795,A -85,B 0,C 180,E1 -14977.239,E2 -14977.239} C_VEL
LIN {X 0,Y 326.58,Z 399.802,A -85,B 0,C 180,E1 -14981.132,E2 -14981.132} C_VEL
LIN {X 0,Y 326.588,Z 399.801,A -85,B 0,C 180,E1 -14984.753,E2 -14984.753} C_VEL
LIN {X 0,Y 326.625,Z 399.798,A -85,B 0,C 180,E1 -14988.162,E2 -14988.162} C_VEL
LIN {X 0,Y 326.64,Z 399.799,A -85,B 0,C 180,E1 -14991.394,E2 -14991.394} C_VEL
LIN {X 0,Y 326.459,Z 399.82,A -85,B 0,C 180,E1 -14994.461,E2 -14994.461} C_VEL
LIN {X 0,Y 326.217,Z 399.853,A -85,B 0,C 180,E1 -14997.412,E2 -14997.412} C_VEL
LIN {X 0,Y 326.089,Z 401.053,A -85,B 0,C 180,E1 -14999.553,E2 -14999.553} C_VEL
LIN {X 0,Y 325.946,Z 403.985,A -85,B 0,C 180,E1 -15003.077,E2 -15003.077} C_VEL
LIN {X 0,Y 325.868,Z 406.416,A -85,B 0,C 180,E1 -15005.809,E2 -15005.809} C_VEL
LIN {X 0,Y 325.824,Z 408.177,A -85,B 0,C 180,E1 -15007.735,E2 -15007.735} C_VEL
LIN {X 0,Y 329.978,Z 421.527,A -85,B 0,C 180,E1 -15008.623,E2 -15008.623} C_VEL
LIN {X 0,Y 332.785,Z 432.575,A -85,B 0,C 180,E1 -15009.522,E2 -15009.522} C_VEL
LIN {X 0,Y 334.254,Z 439.947,A -85,B 0,C 180,E1 -15010.207,E2 -15010.207} C_VEL
LIN {X 0,Y 333.247,Z 451.069,A -85,B 0,C 180,E1 -15011.239,E2 -15011.239} C_VEL
LIN {X 0,Y 332.206,Z 460.985,A -85,B 0,C 180,E1 -15012.394,E2 -15012.394} C_VEL
LIN {X 0,Y 331.066,Z 469.942,A -85,B 0,C 180,E1 -15013.664,E2 -15013.664} C_VEL
LIN {X 0,Y 329.759,Z 478.747,A -85,B 0,C 180,E1 -15015.182,E2 -15015.182} C_VEL
LIN {X 0,Y 328.582,Z 487.321,A -85,B 0,C 180,E1 -15017.022,E2 -15017.022} C_VEL
LIN {X 0,Y 327.531,Z 494.155,A -85,B 0,C 180,E1 -15018.865,E2 -15018.865} C_VEL
LIN {X 0,Y 326.703,Z 499.622,A -85,B 0,C 180,E1 -15020.715,E2 -15020.715} C_VEL
LIN {X 0,Y 326.016,Z 504.661,A -85,B 0,C 180,E1 -15022.951,E2 -15022.951} C_VEL
LIN {X 0,Y 325.521,Z 508.022,A -85,B 0,C 180,E1 -15025.046,E2 -15025.046} C_VEL
LIN {X 0,Y 325.461,Z 509.401,A -85,B 0,C 180,E1 -15026.286,E2 -15026.286} C_VEL
LIN {X 0,Y 325.386,Z 510.383,A -85,B 0,C 180,E1 -15027.524,E2 -15027.524} C_VEL
LIN {X 0,Y 325.232,Z 511.223,A -85,B 0,C 180,E1 -15030,E2 -15030} C_VEL
LIN {X 0,Y 325.382,Z 510.449,A -85,B 0,C 180,E1 -15032.476,E2 -15032.476} C_VEL
LIN {X 0,Y 325.445,Z 509.492,A -85,B 0,C 180,E1 -15033.715,E2 -15033.715} C_VEL
LIN {X 0,Y 325.518,Z 508.152,A -85,B 0,C 180,E1 -15034.954,E2 -15034.954} C_VEL
LIN {X 0,Y 326.007,Z 504.893,A -85,B 0,C 180,E1 -15037.036,E2 -15037.036} C_VEL
LIN {X 0,Y 326.635,Z 499.896,A -85,B 0,C 180,E1 -15039.287,E2 -15039.287} C_VEL
LIN {X 0,Y 327.67,Z 493.491,A -85,B 0,C 180,E1 -15041.443,E2 -15041.443} C_VEL
LIN {X 0,Y 328.696,Z 486.452,A -85,B 0,C 180,E1 -15043.288,E2 -15043.288} C_VEL
LIN {X 0,Y 330.041,Z 477.67,A -85,B 0,C 180,E1 -15045.121,E2 -15045.121} C_VEL
LIN {X 0,Y 331.326,Z 468.652,A -85,B 0,C 180,E1 -15046.64,E2 -15046.64} C_VEL
LIN {X 0,Y 332.434,Z 458.712,A -85,B 0,C 180,E1 -15048.005,E2 -15048.005} C_VEL
LIN {X 0,Y 333.671,Z 447.542,A -85,B 0,C 180,E1 -15049.215,E2 -15049.215} C_VEL
LIN {X 0,Y 334.198,Z 439.146,A -85,B 0,C 180,E1 -15049.972,E2 -15049.972} C_VEL
LIN {X 0,Y 331.678,Z 427.876,A -85,B 0,C 180,E1 -15050.988,E2 -15050.988} C_VEL
LIN {X 0,Y 328.155,Z 415.509,A -85,B 0,C 180,E1 -15051.914,E2 -15051.914} C_VEL
LIN {X 0,Y 325.811,Z 408.12,A -85,B 0,C 180,E1 -15052.391,E2 -15052.391} C_VEL
LIN {X 0,Y 325.898,Z 405.269,A -85,B 0,C 180,E1 -15055.55,E2 -15055.55} C_VEL
LIN {X 0,Y 326.001,Z 402.91,A -85,B 0,C 180,E1 -15058.313,E2 -15058.313} C_VEL
LIN {X 0,Y 326.112,Z 400.58,A -85,B 0,C 180,E1 -15061.146,E2 -15061.146} C_VEL
LIN {X 0,Y 326.228,Z 399.851,A -85,B 0,C 180,E1 -15062.84,E2 -15062.84} C_VEL
LIN {X 0,Y 326.459,Z 399.818,A -85,B 0,C 180,E1 -15065.539,E2 -15065.539} C_VEL
LIN {X 0,Y 326.595,Z 399.805,A -85,B 0,C 180,E1 -15068.613,E2 -15068.613} C_VEL
LIN {X 0,Y 326.579,Z 399.803,A -85,B 0,C 180,E1 -15071.846,E2 -15071.846} C_VEL
LIN {X 0,Y 326.53,Z 399.808,A -85,B 0,C 180,E1 -15075.257,E2 -15075.257} C_VEL
LIN {X 0,Y 326.581,Z 399.803,A -85,B 0,C 180,E1 -15078.869,E2 -15078.869} C_VEL
LIN {X 0,Y 326.633,Z 399.797,A -85,B 0,C 180,E1 -15082.761,E2 -15082.761} C_VEL
LIN {X 0,Y 326.611,Z 399.801,A -85,B 0,C 180,E1 -15085.981,E2 -15085.981} C_VEL
LIN {X 0,Y 326.579,Z 399.799,A -85,B 0,C 180,E1 -15088.107,E2 -15088.107} C_VEL
LIN {X 0,Y 325.902,Z 399.887,A -85,B 0,C 180,E1 -15089.138,E2 -15089.138} C_VEL
LIN {X 0,Y 323.05,Z 400.242,A -85,B 0,C 180,E1 -15090.815,E2 -15090.815} C_VEL
LIN {X 0,Y 320.665,Z 400.543,A -85,B 0,C 180,E1 -15092.175,E2 -15092.175} C_VEL
LIN {X 0,Y 319.676,Z 400.663,A -85,B 0,C 180,E1 -15093.227,E2 -15093.227} C_VEL
LIN {X 0,Y 319.613,Z 400.671,A -85,B 0,C 180,E1 -15093.583,E2 -15093.583} C_VEL
LIN {X 0,Y 319.588,Z 400.674,A -85,B 0,C 180,E1 -15097.461,E2 -15097.461} C_VEL
LIN {X 0,Y 319.692,Z 400.66,A -85,B 0,C 180,E1 -15100.962,E2 -15100.962} C_VEL
LIN {X 0,Y 319.735,Z 400.655,A -85,B 0,C 180,E1 -15105.276,E2 -15105.276} C_VEL
LIN {X 0,Y 319.755,Z 400.657,A -85,B 0,C 180,E1 -15109.873,E2 -15109.873} C_VEL
LIN {X 0,Y 319.941,Z 400.634,A -85,B 0,C 180,E1 -15113.694,E2 -15113.694} C_VEL
LIN {X 0,Y 319.993,Z 400.627,A -85,B 0,C 180,E1 -15117.482,E2 -15117.482} C_VEL
LIN {X 0,Y 320.154,Z 400.606,A -85,B 0,C 180,E1 -15120,E2 -15120} C_VEL
LIN {X 0,Y 319.994,Z 400.624,A -85,B 0,C 180,E1 -15122.518,E2 -15122.518} C_VEL
LIN {X 0,Y 319.956,Z 400.628,A -85,B 0,C 180,E1 -15126.305,E2 -15126.305} C_VEL
LIN {X 0,Y 319.847,Z 400.642,A -85,B 0,C 180,E1 -15128.848,E2 -15128.848} C_VEL
LIN {X 0,Y 319.689,Z 400.661,A -85,B 0,C 180,E1 -15132.7,E2 -15132.7} C_VEL
LIN {X 0,Y 319.703,Z 400.663,A -85,B 0,C 180,E1 -15135.295,E2 -15135.295} C_VEL
LIN {X 0,Y 319.678,Z 400.666,A -85,B 0,C 180,E1 -15139.255,E2 -15139.255} C_VEL
LIN {X 0,Y 319.574,Z 400.68,A -85,B 0,C 180,E1 -15143.319,E2 -15143.319} C_VEL
LIN {X 0,Y 319.637,Z 400.668,A -85,B 0,C 180,E1 -15146.088,E2 -15146.088} C_VEL
LIN {X 0,Y 319.583,Z 400.677,A -85,B 0,C 180,E1 -15148.934,E2 -15148.934} C_VEL
LIN {X 0,Y 319.534,Z 400.681,A -85,B 0,C 180,E1 -15151.862,E2 -15151.862} C_VEL
LIN {X 0,Y 319.583,Z 400.676,A -85,B 0,C 180,E1 -15155.543,E2 -15155.543} C_VEL
LIN {X 0,Y 319.56,Z 400.68,A -85,B 0,C 180,E1 -15158.01,E2 -15158.01} C_VEL
LIN {X 0,Y 319.55,Z 400.686,A -85,B 0,C 180,E1 -15160.867,E2 -15160.867} C_VEL
LIN {X 0,Y 320.443,Z 405.473,A -85,B 0,C 180,E1 -15164.574,E2 -15164.574} C_VEL
LIN {X 0,Y 321.351,Z 410.306,A -85,B 0,C 180,E1 -15168.038,E2 -15168.038} C_VEL
LIN {X 0,Y 322.278,Z 415.817,A -85,B 0,C 180,E1 -15171.726,E2 -15171.726} C_VEL
LIN {X 0,Y 322.356,Z 419.387,A -85,B 0,C 180,E1 -15173.938,E2 -15173.938} C_VEL
LIN {X 0,Y 321.65,Z 424.413,A -85,B 0,C 180,E1 -15176.89,E2 -15176.89} C_VEL
LIN {X 0,Y 320.592,Z 432.058,A -85,B 0,C 180,E1 -15181.268,E2 -15181.268} C_VEL
LIN {X 0,Y 319.708,Z 439.225,A -85,B 0,C 180,E1 -15185.312,E2 -15185.312} C_VEL
LIN {X 0,Y 319.369,Z 442.483,A -85,B 0,C 180,E1 -15187.142,E2 -15187.142} C_VEL
LIN {X 0,Y 322.036,Z 455.991,A -85,B 0,C 180,E1 -15187.873,E2 -15187.873} C_VEL
LIN {X 0,Y 323.807,Z 468.468,A -85,B 0,C 180,E1 -15188.757,E2 -15188.757} C_VEL
LIN {X 0,Y 324.862,Z 479.8,A -85,B 0,C 180,E1 -15189.748,E2 -15189.748} C_VEL
LIN {X 0,Y 325.306,Z 488.064,A -85,B 0,C 180,E1 -15190.599,E2 -15190.599} C_VEL
LIN {X 0,Y 323.722,Z 499.891,A -85,B 0,C 180,E1 -15191.979,E2 -15191.979} C_VEL
LIN {X 0,Y 322.293,Z 510.411,A -85,B 0,C 180,E1 -15193.532,E2 -15193.532} C_VEL
LIN {X 0,Y 321.171,Z 518.939,A -85,B 0,C 180,E1 -15195.101,E2 -15195.101} C_VEL
LIN {X 0,Y 319.982,Z 527.265,A -85,B 0,C 180,E1 -15196.989,E2 -15196.989} C_VEL
LIN {X 0,Y 319.069,Z 533.984,A -85,B 0,C 180,E1 -15198.887,E2 -15198.887} C_VEL
LIN {X 0,Y 318.389,Z 540.146,A -85,B 0,C 180,E1 -15201.111,E2 -15201.111} C_VEL
LIN {X 0,Y 318.093,Z 544.161,A -85,B 0,C 180,E1 -15203.02,E2 -15203.02} C_VEL
LIN {X 0,Y 317.933,Z 547.13,A -85,B 0,C 180,E1 -15204.927,E2 -15204.927} C_VEL
LIN {X 0,Y 317.916,Z 548.546,A -85,B 0,C 180,E1 -15206.197,E2 -15206.197} C_VEL
LIN {X 0,Y 317.951,Z 550.177,A -85,B 0,C 180,E1 -15208.733,E2 -15208.733} C_VEL
LIN {X 0,Y 318.049,Z 550.401,A -85,B 0,C 180,E1 -15210,E2 -15210} C_VEL
LIN {X 0,Y 317.977,Z 550.176,A -85,B 0,C 180,E1 -15211.266,E2 -15211.266} C_VEL
LIN {X 0,Y 317.915,Z 548.541,A -85,B 0,C 180,E1 -15213.803,E2 -15213.803} C_VEL
LIN {X 0,Y 318.001,Z 545.804,A -85,B 0,C 180,E1 -15215.996,E2 -15215.996} C_VEL
LIN {X 0,Y 318.241,Z 541.57,A -85,B 0,C 180,E1 -15218.253,E2 -15218.253} C_VEL
LIN {X 0,Y 318.758,Z 536.799,A -85,B 0,C 180,E1 -15220.159,E2 -15220.159} C_VEL
LIN {X 0,Y 319.592,Z 529.639,A -85,B 0,C 180,E1 -15222.381,E2 -15222.381} C_VEL
LIN {X 0,Y 320.748,Z 521.888,A -85,B 0,C 180,E1 -15224.271,E2 -15224.271} C_VEL
LIN {X 0,Y 322.023,Z 512.919,A -85,B 0,C 180,E1 -15226.02,E2 -15226.02} C_VEL
LIN {X 0,Y 323.214,Z 503.209,A -85,B 0,C 180,E1 -15227.56,E2 -15227.56} C_VEL
LIN {X 0,Y 324.732,Z 492.258,A -85,B 0,C 180,E1 -15228.944,E2 -15228.944} C_VEL
LIN {X 0,Y 325.309,Z 486.405,A -85,B 0,C 180,E1 -15229.564,E2 -15229.564} C_VEL
LIN {X 0,Y 324.424,Z 474.338,A -85,B 0,C 180,E1 -15230.741,E2 -15230.741} C_VEL
LIN {X 0,Y 322.983,Z 462.036,A -85,B 0,C 180,E1 -15231.71,E2 -15231.71} C_VEL
LIN {X 0,Y 320.778,Z 449.244,A -85,B 0,C 180,E1 -15232.507,E2 -15232.507} C_VEL
LIN {X 0,Y 319.374,Z 442.406,A -85,B 0,C 180,E1 -15232.859,E2 -15232.859} C_VEL
LIN {X 0,Y 320.123,Z 435.55,A -85,B 0,C 180,E1 -15236.747,E2 -15236.747} C_VEL
LIN {X 0,Y 320.925,Z 429.374,A -85,B 0,C 180,E1 -15240.244,E2 -15240.244} C_VEL
LIN {X 0,Y 321.897,Z 422.944,A -85,B 0,C 180,E1 -15243.936,E2 -15243.936} C_VEL
LIN {X 0,Y 322.464,Z 417.966,A -85,B 0,C 180,E1 -15246.857,E2 -15246.857} C_VEL
LIN {X 0,Y 322.019,Z 414.178,A -85,B 0,C 180,E1 -15249.266,E2 -15249.266} C_VEL
LIN {X 0,Y 321.13,Z 409.109,A -85,B 0,C 180,E1 -15252.722,E2 -15252.722} C_VEL
LIN {X 0,Y 320.192,Z 404.059,A -85,B 0,C 180,E1 -15256.413,E2 -15256.413} C_VEL
LIN {X 0,Y 319.56,Z 400.683,A -85,B 0,C 180,E1 -15259.135,E2 -15259.135} C_VEL
LIN {X 0,Y 319.564,Z 400.679,A -85,B 0,C 180,E1 -15262.348,E2 -15262.348} C_VEL
LIN {X 0,Y 319.563,Z 400.681,A -85,B 0,C 180,E1 -15265.124,E2 -15265.124} C_VEL
LIN {X 0,Y 319.568,Z 400.679,A -85,B 0,C 180,E1 -15269.059,E2 -15269.059} C_VEL
LIN {X 0,Y 319.608,Z 400.674,A -85,B 0,C 180,E1 -15272.498,E2 -15272.498} C_VEL
LIN {X 0,Y 319.607,Z 400.672,A -85,B 0,C 180,E1 -15275.304,E2 -15275.304} C_VEL
LIN {X 0,Y 319.6,Z 400.673,A -85,B 0,C 180,E1 -15278.048,E2 -15278.048} C_VEL
LIN {X 0,Y 319.691,Z 400.663,A -85,B 0,C 180,E1 -15280.962,E2 -15280.962} C_VEL
LIN {X 0,Y 319.733,Z 400.656,A -85,B 0,C 180,E1 -15285.276,E2 -15285.276} C_VEL
LIN {X 0,Y 319.763,Z 400.652,A -85,B 0,C 180,E1 -15289.873,E2 -15289.873} C_VEL
LIN {X 0,Y 319.936,Z 400.635,A -85,B 0,C 180,E1 -15292.426,E2 -15292.426} C_VEL
LIN {X 0,Y 319.749,Z 400.655,A -85,B 0,C 180,E1 -15294.956,E2 -15294.956} C_VEL
LIN {X 0,Y 319.993,Z 400.623,A -85,B 0,C 180,E1 -15297.482,E2 -15297.482} C_VEL
LIN {X 0,Y 320.172,Z 400.602,A -85,B 0,C 180,E1 -15300,E2 -15300} C_VEL
LIN {X 0,Y 319.992,Z 400.626,A -85,B 0,C 180,E1 -15302.518,E2 -15302.518} C_VEL
LIN {X 0,Y 319.934,Z 400.631,A -85,B 0,C 180,E1 -15306.667,E2 -15306.667} C_VEL
LIN {X 0,Y 319.761,Z 400.656,A -85,B 0,C 180,E1 -15310.127,E2 -15310.127} C_VEL
LIN {X 0,Y 319.733,Z 400.656,A -85,B 0,C 180,E1 -15314.724,E2 -15314.724} C_VEL
LIN {X 0,Y 319.691,Z 400.66,A -85,B 0,C 180,E1 -15319.038,E2 -15319.038} C_VEL
LIN {X 0,Y 319.564,Z 400.677,A -85,B 0,C 180,E1 -15323.32,E2 -15323.32} C_VEL
LIN {X 0,Y 319.636,Z 400.671,A -85,B 0,C 180,E1 -15326.088,E2 -15326.088} C_VEL
LIN {X 0,Y 319.582,Z 400.674,A -85,B 0,C 180,E1 -15328.935,E2 -15328.935} C_VEL
LIN {X 0,Y 319.534,Z 400.684,A -85,B 0,C 180,E1 -15331.862,E2 -15331.862} C_VEL
LIN {X 0,Y 319.583,Z 400.677,A -85,B 0,C 180,E1 -15335.543,E2 -15335.543} C_VEL
LIN {X 0,Y 319.576,Z 400.678,A -85,B 0,C 180,E1 -15338.008,E2 -15338.008} C_VEL
LIN {X 0,Y 319.528,Z 400.684,A -85,B 0,C 180,E1 -15341.597,E2 -15341.597} C_VEL
LIN {X 0,Y 319.58,Z 400.676,A -85,B 0,C 180,E1 -15345.273,E2 -15345.273} C_VEL
LIN {X 0,Y 319.582,Z 400.674,A -85,B 0,C 180,E1 -15348.72,E2 -15348.72} C_VEL
LIN {X 0,Y 319.551,Z 400.68,A -85,B 0,C 180,E1 -15352.351,E2 -15352.351} C_VEL
LIN {X 0,Y 319.357,Z 400.707,A -85,B 0,C 180,E1 -15355.098,E2 -15355.098} C_VEL
LIN {X 0,Y 319.085,Z 400.872,A -85,B 0,C 180,E1 -15358.088,E2 -15358.088} C_VEL
LIN {X 0,Y 318.969,Z 403.214,A -85,B 0,C 180,E1 -15361.005,E2 -15361.005} C_VEL
LIN {X 0,Y 318.859,Z 406.83,A -85,B 0,C 180,E1 -15365.242,E2 -15365.242} C_VEL
LIN {X 0,Y 318.801,Z 408.627,A -85,B 0,C 180,E1 -15367.216,E2 -15367.216} C_VEL
LIN {X 0,Y 323.089,Z 422.146,A -85,B 0,C 180,E1 -15368.153,E2 -15368.153} C_VEL
LIN {X 0,Y 326.292,Z 434.885,A -85,B 0,C 180,E1 -15369.235,E2 -15369.235} C_VEL
LIN {X 0,Y 327.529,Z 441.863,A -85,B 0,C 180,E1 -15369.921,E2 -15369.921} C_VEL
LIN {X 0,Y 326.422,Z 452.92,A -85,B 0,C 180,E1 -15370.995,E2 -15370.995} C_VEL
LIN {X 0,Y 325.313,Z 462.979,A -85,B 0,C 180,E1 -15372.226,E2 -15372.226} C_VEL
LIN {X 0,Y 324.021,Z 472.311,A -85,B 0,C 180,E1 -15373.622,E2 -15373.622} C_VEL
LIN {X 0,Y 322.727,Z 480.768,A -85,B 0,C 180,E1 -15375.174,E2 -15375.174} C_VEL
LIN {X 0,Y 321.48,Z 488.976,A -85,B 0,C 180,E1 -15377.051,E2 -15377.051} C_VEL
LIN {X 0,Y 320.598,Z 494.588,A -85,B 0,C 180,E1 -15378.621,E2 -15378.621} C_VEL
LIN {X 0,Y 319.693,Z 500.057,A -85,B 0,C 180,E1 -15380.51,E2 -15380.51} C_VEL
LIN {X 0,Y 319.1,Z 504.34,A -85,B 0,C 180,E1 -15382.406,E2 -15382.406} C_VEL
LIN {X 0,Y 318.775,Z 506.607,A -85,B 0,C 180,E1 -15383.671,E2 -15383.671} C_VEL
LIN {X 0,Y 318.468,Z 508.453,A -85,B 0,C 180,E1 -15384.936,E2 -15384.936} C_VEL
LIN {X 0,Y 318.38,Z 509.833,A -85,B 0,C 180,E1 -15386.203,E2 -15386.203} C_VEL
LIN {X 0,Y 318.317,Z 510.815,A -85,B 0,C 180,E1 -15387.469,E2 -15387.469} C_VEL
LIN {X 0,Y 318.156,Z 511.654,A -85,B 0,C 180,E1 -15390,E2 -15390} C_VEL
LIN {X 0,Y 318.298,Z 510.88,A -85,B 0,C 180,E1 -15392.531,E2 -15392.531} C_VEL
LIN {X 0,Y 318.465,Z 508.582,A -85,B 0,C 180,E1 -15395.064,E2 -15395.064} C_VEL
LIN {X 0,Y 318.942,Z 505.569,A -85,B 0,C 180,E1 -15397.059,E2 -15397.059} C_VEL
LIN {X 0,Y 319.433,Z 501.873,A -85,B 0,C 180,E1 -15398.86,E2 -15398.86} C_VEL
LIN {X 0,Y 320.215,Z 496.886,A -85,B 0,C 180,E1 -15400.752,E2 -15400.752} C_VEL
LIN {X 0,Y 321.244,Z 490.6,A -85,B 0,C 180,E1 -15402.637,E2 -15402.637} C_VEL
LIN {X 0,Y 322.493,Z 482.728,A -85,B 0,C 180,E1 -15404.514,E2 -15404.514} C_VEL
LIN {X 0,Y 323.703,Z 474.698,A -85,B 0,C 180,E1 -15406.071,E2 -15406.071} C_VEL
LIN {X 0,Y 325.076,Z 464.892,A -85,B 0,C 180,E1 -15407.619,E2 -15407.619} C_VEL
LIN {X 0,Y 326.148,Z 455.243,A -85,B 0,C 180,E1 -15408.858,E2 -15408.858} C_VEL
LIN {X 0,Y 327.315,Z 444.776,A -85,B 0,C 180,E1 -15409.93,E2 -15409.93} C_VEL
LIN {X 0,Y 327.563,Z 441.45,A -85,B 0,C 180,E1 -15410.224,E2 -15410.224} C_VEL
LIN {X 0,Y 325.262,Z 430.411,A -85,B 0,C 180,E1 -15411.281,E2 -15411.281} C_VEL
LIN {X 0,Y 321.916,Z 418.342,A -85,B 0,C 180,E1 -15412.248,E2 -15412.248} C_VEL
LIN {X 0,Y 318.763,Z 408.539,A -85,B 0,C 180,E1 -15412.936,E2 -15412.936} C_VEL
LIN {X 0,Y 318.88,Z 405.691,A -85,B 0,C 180,E1 -15416.155,E2 -15416.155} C_VEL
LIN {X 0,Y 318.978,Z 403.311,A -85,B 0,C 180,E1 -15418.995,E2 -15418.995} C_VEL
LIN {X 0,Y 319.115,Z 400.963,A -85,B 0,C 180,E1 -15421.909,E2 -15421.909} C_VEL
LIN {X 0,Y 319.436,Z 400.693,A -85,B 0,C 180,E1 -15425.506,E2 -15425.506} C_VEL
LIN {X 0,Y 319.532,Z 400.682,A -85,B 0,C 180,E1 -15428.014,E2 -15428.014} C_VEL
LIN {X 0,Y 319.528,Z 400.681,A -85,B 0,C 180,E1 -15431.597,E2 -15431.597} C_VEL
LIN {X 0,Y 319.491,Z 400.685,A -85,B 0,C 180,E1 -15435.257,E2 -15435.257} C_VEL
LIN {X 0,Y 319.532,Z 400.682,A -85,B 0,C 180,E1 -15438.712,E2 -15438.712} C_VEL
LIN {X 0,Y 319.582,Z 400.679,A -85,B 0,C 180,E1 -15442.344,E2 -15442.344} C_VEL
LIN {X 0,Y 319.564,Z 400.675,A -85,B 0,C 180,E1 -15445.124,E2 -15445.124} C_VEL
LIN {X 0,Y 319.57,Z 400.675,A -85,B 0,C 180,E1 -15449.059,E2 -15449.059} C_VEL
LIN {X 0,Y 319.609,Z 400.673,A -85,B 0,C 180,E1 -15452.498,E2 -15452.498} C_VEL
LIN {X 0,Y 319.613,Z 400.671,A -85,B 0,C 180,E1 -15453.583,E2 -15453.583} C_VEL
LIN {X 0,Y 318.989,Z 400.754,A -85,B 0,C 180,E1 -15454.635,E2 -15454.635} C_VEL
LIN {X 0,Y 316.129,Z 401.112,A -85,B 0,C 180,E1 -15456.346,E2 -15456.346} C_VEL
LIN {X 0,Y 313.676,Z 401.414,A -85,B 0,C 180,E1 -15457.734,E2 -15457.734} C_VEL
LIN {X 0,Y 312.621,Z 401.541,A -85,B 0,C 180,E1 -15458.809,E2 -15458.809} C_VEL
LIN {X 0,Y 312.536,Z 401.55,A -85,B 0,C 180,E1 -15459.174,E2 -15459.174} C_VEL
LIN {X 0,Y 312.642,Z 401.54,A -85,B 0,C 180,E1 -15461.656,E2 -15461.656} C_VEL
LIN {X 0,Y 312.698,Z 401.535,A -85,B 0,C 180,E1 -15465.686,E2 -15465.686} C_VEL
LIN {X 0,Y 312.702,Z 401.534,A -85,B 0,C 180,E1 -15469.642,E2 -15469.642} C_VEL
LIN {X 0,Y 312.897,Z 401.51,A -85,B 0,C 180,E1 -15473.552,E2 -15473.552} C_VEL
LIN {X 0,Y 312.94,Z 401.505,A -85,B 0,C 180,E1 -15477.426,E2 -15477.426} C_VEL
LIN {X 0,Y 313.106,Z 401.484,A -85,B 0,C 180,E1 -15480,E2 -15480} C_VEL
LIN {X 0,Y 312.94,Z 401.503,A -85,B 0,C 180,E1 -15482.574,E2 -15482.574} C_VEL
LIN {X 0,Y 312.915,Z 401.505,A -85,B 0,C 180,E1 -15486.448,E2 -15486.448} C_VEL
LIN {X 0,Y 312.792,Z 401.522,A -85,B 0,C 180,E1 -15489.049,E2 -15489.049} C_VEL
LIN {X 0,Y 312.641,Z 401.54,A -85,B 0,C 180,E1 -15492.991,E2 -15492.991} C_VEL
LIN {X 0,Y 312.642,Z 401.541,A -85,B 0,C 180,E1 -15495.65,E2 -15495.65} C_VEL
LIN {X 0,Y 312.634,Z 401.543,A -85,B 0,C 180,E1 -15499.236,E2 -15499.236} C_VEL
LIN {X 0,Y 312.549,Z 401.551,A -85,B 0,C 180,E1 -15502.789,E2 -15502.789} C_VEL
LIN {X 0,Y 312.606,Z 401.544,A -85,B 0,C 180,E1 -15505.935,E2 -15505.935} C_VEL
LIN {X 0,Y 312.541,Z 401.554,A -85,B 0,C 180,E1 -15509.65,E2 -15509.65} C_VEL
LIN {X 0,Y 312.522,Z 401.556,A -85,B 0,C 180,E1 -15513.689,E2 -15513.689} C_VEL
LIN {X 0,Y 312.529,Z 401.555,A -85,B 0,C 180,E1 -15517.385,E2 -15517.385} C_VEL
LIN {X 0,Y 312.539,Z 401.62,A -85,B 0,C 180,E1 -15520.358,E2 -15520.358} C_VEL
LIN {X 0,Y 313.397,Z 406.367,A -85,B 0,C 180,E1 -15524.142,E2 -15524.142} C_VEL
LIN {X 0,Y 314.332,Z 411.416,A -85,B 0,C 180,E1 -15527.874,E2 -15527.874} C_VEL
LIN {X 0,Y 315.21,Z 416.494,A -85,B 0,C 180,E1 -15531.369,E2 -15531.369} C_VEL
LIN {X 0,Y 315.403,Z 419.534,A -85,B 0,C 180,E1 -15533.338,E2 -15533.338} C_VEL
LIN {X 0,Y 314.833,Z 424.047,A -85,B 0,C 180,E1 -15536.077,E2 -15536.077} C_VEL
LIN {X 0,Y 313.859,Z 430.253,A -85,B 0,C 180,E1 -15539.746,E2 -15539.746} C_VEL
LIN {X 0,Y 312.919,Z 437.459,A -85,B 0,C 180,E1 -15543.946,E2 -15543.946} C_VEL
LIN {X 0,Y 312.377,Z 442.034,A -85,B 0,C 180,E1 -15546.595,E2 -15546.595} C_VEL
LIN {X 0,Y 315.169,Z 455.957,A -85,B 0,C 180,E1 -15547.388,E2 -15547.388} C_VEL
LIN {X 0,Y 316.903,Z 467.833,A -85,B 0,C 180,E1 -15548.257,E2 -15548.257} C_VEL
LIN {X 0,Y 317.95,Z 479.356,A -85,B 0,C 180,E1 -15549.288,E2 -15549.288} C_VEL
LIN {X 0,Y 318.404,Z 489.067,A -85,B 0,C 180,E1 -15550.329,E2 -15550.329} C_VEL
LIN {X 0,Y 316.776,Z 500.641,A -85,B 0,C 180,E1 -15551.737,E2 -15551.737} C_VEL
LIN {X 0,Y 315.274,Z 511.061,A -85,B 0,C 180,E1 -15553.354,E2 -15553.354} C_VEL
LIN {X 0,Y 314.298,Z 518.508,A -85,B 0,C 180,E1 -15554.767,E2 -15554.767} C_VEL
LIN {X 0,Y 313.01,Z 526.83,A -85,B 0,C 180,E1 -15556.694,E2 -15556.694} C_VEL
LIN {X 0,Y 312.048,Z 533.549,A -85,B 0,C 180,E1 -15558.634,E2 -15558.634} C_VEL
LIN {X 0,Y 311.361,Z 539.714,A -85,B 0,C 180,E1 -15560.909,E2 -15560.909} C_VEL
LIN {X 0,Y 311.021,Z 543.727,A -85,B 0,C 180,E1 -15562.861,E2 -15562.861} C_VEL
LIN {X 0,Y 310.85,Z 546.697,A -85,B 0,C 180,E1 -15564.811,E2 -15564.811} C_VEL
LIN {X 0,Y 310.846,Z 548.115,A -85,B 0,C 180,E1 -15566.111,E2 -15566.111} C_VEL
LIN {X 0,Y 310.858,Z 549.745,A -85,B 0,C 180,E1 -15568.704,E2 -15568.704} C_VEL
LIN {X 0,Y 310.96,Z 549.97,A -85,B 0,C 180,E1 -15570,E2 -15570} C_VEL
LIN {X 0,Y 310.883,Z 549.744,A -85,B 0,C 180,E1 -15571.295,E2 -15571.295} C_VEL
LIN {X 0,Y 310.845,Z 548.109,A -85,B 0,C 180,E1 -15573.889,E2 -15573.889} C_VEL
LIN {X 0,Y 310.899,Z 545.648,A -85,B 0,C 180,E1 -15575.935,E2 -15575.935} C_VEL
LIN {X 0,Y 311.064,Z 542.464,A -85,B 0,C 180,E1 -15577.791,E2 -15577.791} C_VEL
LIN {X 0,Y 311.521,Z 538.077,A -85,B 0,C 180,E1 -15579.741,E2 -15579.741} C_VEL
LIN {X 0,Y 312.154,Z 532.492,A -85,B 0,C 180,E1 -15581.691,E2 -15581.691} C_VEL
LIN {X 0,Y 313.213,Z 525.543,A -85,B 0,C 180,E1 -15583.627,E2 -15583.627} C_VEL
LIN {X 0,Y 314.548,Z 516.857,A -85,B 0,C 180,E1 -15585.552,E2 -15585.552} C_VEL
LIN {X 0,Y 315.707,Z 507.948,A -85,B 0,C 180,E1 -15587.155,E2 -15587.155} C_VEL
LIN {X 0,Y 317.132,Z 498.193,A -85,B 0,C 180,E1 -15588.576,E2 -15588.576} C_VEL
LIN {X 0,Y 318.478,Z 487.521,A -85,B 0,C 180,E1 -15589.833,E2 -15589.833} C_VEL
LIN {X 0,Y 317.604,Z 475.029,A -85,B 0,C 180,E1 -15591.111,E2 -15591.111} C_VEL
LIN {X 0,Y 316.207,Z 462.625,A -85,B 0,C 180,E1 -15592.132,E2 -15592.132} C_VEL
LIN {X 0,Y 314.01,Z 449.66,A -85,B 0,C 180,E1 -15592.985,E2 -15592.985} C_VEL
LIN {X 0,Y 312.35,Z 441.966,A -85,B 0,C 180,E1 -15593.391,E2 -15593.391} C_VEL
LIN {X 0,Y 313.192,Z 435.139,A -85,B 0,C 180,E1 -15597.388,E2 -15597.388} C_VEL
LIN {X 0,Y 314.033,Z 428.985,A -85,B 0,C 180,E1 -15600.98,E2 -15600.98} C_VEL
LIN {X 0,Y 314.936,Z 423.316,A -85,B 0,C 180,E1 -15604.343,E2 -15604.343} C_VEL
LIN {X 0,Y 315.462,Z 418.954,A -85,B 0,C 180,E1 -15606.979,E2 -15606.979} C_VEL
LIN {X 0,Y 314.777,Z 413.83,A -85,B 0,C 180,E1 -15610.352,E2 -15610.352} C_VEL
LIN {X 0,Y 313.794,Z 408.428,A -85,B 0,C 180,E1 -15614.217,E2 -15614.217} C_VEL
LIN {X 0,Y 312.916,Z 403.781,A -85,B 0,C 180,E1 -15617.831,E2 -15617.831} C_VEL
LIN {X 0,Y 312.516,Z 401.561,A -85,B 0,C 180,E1 -15619.809,E2 -15619.809} C_VEL
LIN {X 0,Y 312.538,Z 401.553,A -85,B 0,C 180,E1 -15624.05,E2 -15624.05} C_VEL
LIN {X 0,Y 312.506,Z 401.559,A -85,B 0,C 180,E1 -15627.334,E2 -15627.334} C_VEL
LIN {X 0,Y 312.546,Z 401.552,A -85,B 0,C 180,E1 -15631.279,E2 -15631.279} C_VEL
LIN {X 0,Y 312.587,Z 401.55,A -85,B 0,C 180,E1 -15634.711,E2 -15634.711} C_VEL
LIN {X 0,Y 312.59,Z 401.545,A -85,B 0,C 180,E1 -15637.529,E2 -15637.529} C_VEL
LIN {X 0,Y 312.641,Z 401.539,A -85,B 0,C 180,E1 -15641.657,E2 -15641.657} C_VEL
LIN {X 0,Y 312.697,Z 401.532,A -85,B 0,C 180,E1 -15645.686,E2 -15645.686} C_VEL
LIN {X 0,Y 312.707,Z 401.531,A -85,B 0,C 180,E1 -15649.642,E2 -15649.642} C_VEL
LIN {X 0,Y 312.875,Z 401.513,A -85,B 0,C 180,E1 -15652.254,E2 -15652.254} C_VEL
LIN {X 0,Y 312.72,Z 401.531,A -85,B 0,C 180,E1 -15654.842,E2 -15654.842} C_VEL
LIN {X 0,Y 312.994,Z 401.497,A -85,B 0,C 180,E1 -15658.713,E2 -15658.713} C_VEL
LIN {X 0,Y 313.123,Z 401.48,A -85,B 0,C 180,E1 -15660,E2 -15660} C_VEL
LIN {X 0,Y 312.939,Z 401.504,A -85,B 0,C 180,E1 -15662.574,E2 -15662.574} C_VEL
LIN {X 0,Y 312.897,Z 401.508,A -85,B 0,C 180,E1 -15666.651,E2 -15666.651} C_VEL
LIN {X 0,Y 312.79,Z 401.52,A -85,B 0,C 180,E1 -15669.049,E2 -15669.049} C_VEL
LIN {X 0,Y 312.637,Z 401.538,A -85,B 0,C 180,E1 -15672.991,E2 -15672.991} C_VEL
LIN {X 0,Y 312.641,Z 401.54,A -85,B 0,C 180,E1 -15675.65,E2 -15675.65} C_VEL
LIN {X 0,Y 312.632,Z 401.539,A -85,B 0,C 180,E1 -15679.236,E2 -15679.236} C_VEL
LIN {X 0,Y 312.53,Z 401.553,A -85,B 0,C 180,E1 -15682.781,E2 -15682.781} C_VEL
LIN {X 0,Y 312.604,Z 401.548,A -85,B 0,C 180,E1 -15685.936,E2 -15685.936} C_VEL
LIN {X 0,Y 312.54,Z 401.554,A -85,B 0,C 180,E1 -15689.651,E2 -15689.651} C_VEL
LIN {X 0,Y 312.522,Z 401.555,A -85,B 0,C 180,E1 -15693.689,E2 -15693.689} C_VEL
LIN {X 0,Y 312.54,Z 401.551,A -85,B 0,C 180,E1 -15697.383,E2 -15697.383} C_VEL
LIN {X 0,Y 312.492,Z 401.557,A -85,B 0,C 180,E1 -15700.709,E2 -15700.709} C_VEL
LIN {X 0,Y 312.522,Z 401.555,A -85,B 0,C 180,E1 -15704.197,E2 -15704.197} C_VEL
LIN {X 0,Y 312.551,Z 401.553,A -85,B 0,C 180,E1 -15707.905,E2 -15707.905} C_VEL
LIN {X 0,Y 312.522,Z 401.558,A -85,B 0,C 180,E1 -15711.914,E2 -15711.914} C_VEL
LIN {X 0,Y 312.403,Z 401.572,A -85,B 0,C 180,E1 -15714.203,E2 -15714.203} C_VEL
LIN {X 0,Y 312.079,Z 401.614,A -85,B 0,C 180,E1 -15717.284,E2 -15717.284} C_VEL
LIN {X 0,Y 312.039,Z 402.481,A -85,B 0,C 180,E1 -15718.856,E2 -15718.856} C_VEL
LIN {X 0,Y 311.923,Z 404.807,A -85,B 0,C 180,E1 -15721.761,E2 -15721.761} C_VEL
LIN {X 0,Y 311.848,Z 407.248,A -85,B 0,C 180,E1 -15724.647,E2 -15724.647} C_VEL
LIN {X 0,Y 311.751,Z 409.022,A -85,B 0,C 180,E1 -15726.651,E2 -15726.651} C_VEL
LIN {X 0,Y 316.586,Z 424.09,A -85,B 0,C 180,E1 -15727.766,E2 -15727.766} C_VEL
LIN {X 0,Y 319.512,Z 435.859,A -85,B 0,C 180,E1 -15728.816,E2 -15728.816} C_VEL
LIN {X 0,Y 320.813,Z 442.306,A -85,B 0,C 180,E1 -15729.481,E2 -15729.481} C_VEL
LIN {X 0,Y 319.731,Z 453.356,A -85,B 0,C 180,E1 -15730.582,E2 -15730.582} C_VEL
LIN {X 0,Y 318.558,Z 463.617,A -85,B 0,C 180,E1 -15731.865,E2 -15731.865} C_VEL
LIN {X 0,Y 317.236,Z 472.746,A -85,B 0,C 180,E1 -15733.262,E2 -15733.262} C_VEL
LIN {X 0,Y 315.876,Z 481.203,A -85,B 0,C 180,E1 -15734.845,E2 -15734.845} C_VEL
LIN {X 0,Y 314.594,Z 489.409,A -85,B 0,C 180,E1 -15736.763,E2 -15736.763} C_VEL
LIN {X 0,Y 313.67,Z 495.02,A -85,B 0,C 180,E1 -15738.367,E2 -15738.367} C_VEL
LIN {X 0,Y 312.706,Z 500.49,A -85,B 0,C 180,E1 -15740.296,E2 -15740.296} C_VEL
LIN {X 0,Y 312.095,Z 504.772,A -85,B 0,C 180,E1 -15742.235,E2 -15742.235} C_VEL
LIN {X 0,Y 311.749,Z 507.039,A -85,B 0,C 180,E1 -15743.528,E2 -15743.528} C_VEL
LIN {X 0,Y 311.419,Z 508.885,A -85,B 0,C 180,E1 -15744.821,E2 -15744.821} C_VEL
LIN {X 0,Y 311.301,Z 510.266,A -85,B 0,C 180,E1 -15746.117,E2 -15746.117} C_VEL
LIN {X 0,Y 311.233,Z 511.247,A -85,B 0,C 180,E1 -15747.412,E2 -15747.412} C_VEL
LIN {X 0,Y 311.082,Z 512.085,A -85,B 0,C 180,E1 -15750,E2 -15750} C_VEL
LIN {X 0,Y 311.113,Z 511.894,A -85,B 0,C 180,E1 -15751.295,E2 -15751.295} C_VEL
LIN {X 0,Y 311.214,Z 511.312,A -85,B 0,C 180,E1 -15752.589,E2 -15752.589} C_VEL
LIN {X 0,Y 311.416,Z 509.013,A -85,B 0,C 180,E1 -15755.179,E2 -15755.179} C_VEL
LIN {X 0,Y 311.877,Z 506.221,A -85,B 0,C 180,E1 -15757.084,E2 -15757.084} C_VEL
LIN {X 0,Y 312.428,Z 502.304,A -85,B 0,C 180,E1 -15759.06,E2 -15759.06} C_VEL
LIN {X 0,Y 313.261,Z 497.316,A -85,B 0,C 180,E1 -15760.994,E2 -15760.994} C_VEL
LIN {X 0,Y 314.347,Z 491.028,A -85,B 0,C 180,E1 -15762.919,E2 -15762.919} C_VEL
LIN {X 0,Y 315.614,Z 483.158,A -85,B 0,C 180,E1 -15764.838,E2 -15764.838} C_VEL
LIN {X 0,Y 317.235,Z 473.354,A -85,B 0,C 180,E1 -15766.739,E2 -15766.739} C_VEL
LIN {X 0,Y 318.544,Z 463.493,A -85,B 0,C 180,E1 -15768.263,E2 -15768.263} C_VEL
LIN {X 0,Y 319.766,Z 452.866,A -85,B 0,C 180,E1 -15769.583,E2 -15769.583} C_VEL
LIN {X 0,Y 320.816,Z 443.446,A -85,B 0,C 180,E1 -15770.519,E2 -15770.519} C_VEL
LIN {X 0,Y 319.36,Z 435.113,A -85,B 0,C 180,E1 -15771.366,E2 -15771.366} C_VEL
LIN {X 0,Y 316.044,Z 422.366,A -85,B 0,C 180,E1 -15772.486,E2 -15772.486} C_VEL
LIN {X 0,Y 311.738,Z 408.983,A -85,B 0,C 180,E1 -15773.477,E2 -15773.477} C_VEL
LIN {X 0,Y 311.853,Z 406.114,A -85,B 0,C 180,E1 -15776.791,E2 -15776.791} C_VEL
LIN {X 0,Y 311.972,Z 403.715,A -85,B 0,C 180,E1 -15779.71,E2 -15779.71} C_VEL
LIN {X 0,Y 312.092,Z 401.612,A -85,B 0,C 180,E1 -15782.715,E2 -15782.715} C_VEL
LIN {X 0,Y 312.428,Z 401.568,A -85,B 0,C 180,E1 -15785.922,E2 -15785.922} C_VEL
LIN {X 0,Y 312.496,Z 401.558,A -85,B 0,C 180,E1 -15789.03,E2 -15789.03} C_VEL
LIN {X 0,Y 312.493,Z 401.562,A -85,B 0,C 180,E1 -15792.432,E2 -15792.432} C_VEL
LIN {X 0,Y 312.461,Z 401.563,A -85,B 0,C 180,E1 -15796.035,E2 -15796.035} C_VEL
LIN {X 0,Y 312.507,Z 401.557,A -85,B 0,C 180,E1 -15799.875,E2 -15799.875} C_VEL
LIN {X 0,Y 312.542,Z 401.553,A -85,B 0,C 180,E1 -15802.617,E2 -15802.617} C_VEL
LIN {X 0,Y 312.523,Z 401.558,A -85,B 0,C 180,E1 -15806.311,E2 -15806.311} C_VEL
LIN {X 0,Y 312.541,Z 401.555,A -85,B 0,C 180,E1 -15810.349,E2 -15810.349} C_VEL
LIN {X 0,Y 312.606,Z 401.548,A -85,B 0,C 180,E1 -15814.065,E2 -15814.065} C_VEL
LIN {X 0,Y 312.568,Z 401.549,A -85,B 0,C 180,E1 -15817.527,E2 -15817.527} C_VEL
LIN {X 0,Y 312.536,Z 401.55,A -85,B 0,C 180,E1 -15819.174,E2 -15819.174} C_VEL
LIN {X 0,Y 311.87,Z 401.637,A -85,B 0,C 180,E1 -15820.25,E2 -15820.25} C_VEL
LIN {X 0,Y 309.029,Z 401.993,A -85,B 0,C 180,E1 -15822.002,E2 -15822.002} C_VEL
LIN {X 0,Y 306.656,Z 402.287,A -85,B 0,C 180,E1 -15823.424,E2 -15823.424} C_VEL
LIN {X 0,Y 305.688,Z 402.406,A -85,B 0,C 180,E1 -15824.524,E2 -15824.524} C_VEL
LIN {X 0,Y 305.636,Z 402.411,A -85,B 0,C 180,E1 -15824.896,E2 -15824.896} C_VEL
LIN {X 0,Y 305.639,Z 402.412,A -85,B 0,C 180,E1 -15829.4,E2 -15829.4} C_VEL
LIN {X 0,Y 305.776,Z 402.397,A -85,B 0,C 180,E1 -15832.073,E2 -15832.073} C_VEL
LIN {X 0,Y 305.688,Z 402.405,A -85,B 0,C 180,E1 -15834.723,E2 -15834.723} C_VEL
LIN {X 0,Y 305.96,Z 402.372,A -85,B 0,C 180,E1 -15838.684,E2 -15838.684} C_VEL
LIN {X 0,Y 305.96,Z 402.374,A -85,B 0,C 180,E1 -15841.316,E2 -15841.316} C_VEL
LIN {X 0,Y 305.857,Z 402.384,A -85,B 0,C 180,E1 -15846.597,E2 -15846.597} C_VEL
LIN {X 0,Y 305.74,Z 402.402,A -85,B 0,C 180,E1 -15849.26,E2 -15849.26} C_VEL
LIN {X 0,Y 305.596,Z 402.42,A -85,B 0,C 180,E1 -15853.296,E2 -15853.296} C_VEL
LIN {X 0,Y 305.598,Z 402.416,A -85,B 0,C 180,E1 -15856.02,E2 -15856.02} C_VEL
LIN {X 0,Y 305.58,Z 402.423,A -85,B 0,C 180,E1 -15859.445,E2 -15859.445} C_VEL
LIN {X 0,Y 305.494,Z 402.432,A -85,B 0,C 180,E1 -15863.041,E2 -15863.041} C_VEL
LIN {X 0,Y 305.535,Z 402.425,A -85,B 0,C 180,E1 -15866.221,E2 -15866.221} C_VEL
LIN {X 0,Y 305.492,Z 402.433,A -85,B 0,C 180,E1 -15869.047,E2 -15869.047} C_VEL
LIN {X 0,Y 305.445,Z 402.436,A -85,B 0,C 180,E1 -15871.952,E2 -15871.952} C_VEL
LIN {X 0,Y 305.465,Z 402.434,A -85,B 0,C 180,E1 -15875.113,E2 -15875.113} C_VEL
LIN {X 0,Y 305.476,Z 402.435,A -85,B 0,C 180,E1 -15879.255,E2 -15879.255} C_VEL
LIN {X 0,Y 305.498,Z 402.628,A -85,B 0,C 180,E1 -15879.888,E2 -15879.888} C_VEL
LIN {X 0,Y 306.321,Z 406.965,A -85,B 0,C 180,E1 -15883.496,E2 -15883.496} C_VEL
LIN {X 0,Y 307.176,Z 411.64,A -85,B 0,C 180,E1 -15887.066,E2 -15887.066} C_VEL
LIN {X 0,Y 308.091,Z 416.962,A -85,B 0,C 180,E1 -15890.859,E2 -15890.859} C_VEL
LIN {X 0,Y 308.392,Z 419.997,A -85,B 0,C 180,E1 -15892.904,E2 -15892.904} C_VEL
LIN {X 0,Y 307.982,Z 423.706,A -85,B 0,C 180,E1 -15895.236,E2 -15895.236} C_VEL
LIN {X 0,Y 306.987,Z 429.858,A -85,B 0,C 180,E1 -15898.995,E2 -15898.995} C_VEL
LIN {X 0,Y 306.123,Z 435.967,A -85,B 0,C 180,E1 -15902.667,E2 -15902.667} C_VEL
LIN {X 0,Y 305.38,Z 441.58,A -85,B 0,C 180,E1 -15906.015,E2 -15906.015} C_VEL
LIN {X 0,Y 308.308,Z 455.777,A -85,B 0,C 180,E1 -15906.871,E2 -15906.871} C_VEL
LIN {X 0,Y 310.053,Z 467.869,A -85,B 0,C 180,E1 -15907.788,E2 -15907.788} C_VEL
LIN {X 0,Y 311.055,Z 478.912,A -85,B 0,C 180,E1 -15908.807,E2 -15908.807} C_VEL
LIN {X 0,Y 311.654,Z 488.634,A -85,B 0,C 180,E1 -15909.885,E2 -15909.885} C_VEL
LIN {X 0,Y 310.019,Z 500.21,A -85,B 0,C 180,E1 -15911.324,E2 -15911.324} C_VEL
LIN {X 0,Y 308.619,Z 509.546,A -85,B 0,C 180,E1 -15912.78,E2 -15912.78} C_VEL
LIN {X 0,Y 307.435,Z 518.076,A -85,B 0,C 180,E1 -15914.418,E2 -15914.418} C_VEL
LIN {X 0,Y 306.069,Z 526.398,A -85,B 0,C 180,E1 -15916.387,E2 -15916.387} C_VEL
LIN {X 0,Y 305.022,Z 533.114,A -85,B 0,C 180,E1 -15918.369,E2 -15918.369} C_VEL
LIN {X 0,Y 304.309,Z 539.28,A -85,B 0,C 180,E1 -15920.696,E2 -15920.696} C_VEL
LIN {X 0,Y 303.948,Z 543.294,A -85,B 0,C 180,E1 -15922.694,E2 -15922.694} C_VEL
LIN {X 0,Y 303.77,Z 546.265,A -85,B 0,C 180,E1 -15924.69,E2 -15924.69} C_VEL
LIN {X 0,Y 303.755,Z 547.683,A -85,B 0,C 180,E1 -15926.02,E2 -15926.02} C_VEL
LIN {X 0,Y 303.766,Z 549.313,A -85,B 0,C 180,E1 -15928.674,E2 -15928.674} C_VEL
LIN {X 0,Y 303.871,Z 549.538,A -85,B 0,C 180,E1 -15930,E2 -15930} C_VEL
LIN {X 0,Y 303.789,Z 549.311,A -85,B 0,C 180,E1 -15931.325,E2 -15931.325} C_VEL
LIN {X 0,Y 303.754,Z 547.676,A -85,B 0,C 180,E1 -15933.98,E2 -15933.98} C_VEL
LIN {X 0,Y 303.831,Z 545.412,A -85,B 0,C 180,E1 -15935.93,E2 -15935.93} C_VEL
LIN {X 0,Y 304.016,Z 542.03,A -85,B 0,C 180,E1 -15937.973,E2 -15937.973} C_VEL
LIN {X 0,Y 304.481,Z 537.64,A -85,B 0,C 180,E1 -15939.969,E2 -15939.969} C_VEL
LIN {X 0,Y 305.162,Z 532.056,A -85,B 0,C 180,E1 -15941.963,E2 -15941.963} C_VEL
LIN {X 0,Y 306.293,Z 525.107,A -85,B 0,C 180,E1 -15943.941,E2 -15943.941} C_VEL
LIN {X 0,Y 307.424,Z 518.018,A -85,B 0,C 180,E1 -15945.582,E2 -15945.582} C_VEL
LIN {X 0,Y 308.619,Z 509.472,A -85,B 0,C 180,E1 -15947.22,E2 -15947.22} C_VEL
LIN {X 0,Y 310.012,Z 500.114,A -85,B 0,C 180,E1 -15948.676,E2 -15948.676} C_VEL
LIN {X 0,Y 311.625,Z 488.518,A -85,B 0,C 180,E1 -15950.116,E2 -15950.116} C_VEL
LIN {X 0,Y 310.925,Z 476.818,A -85,B 0,C 180,E1 -15951.39,E2 -15951.39} C_VEL
LIN {X 0,Y 309.636,Z 464.548,A -85,B 0,C 180,E1 -15952.469,E2 -15952.469} C_VEL
LIN {X 0,Y 307.431,Z 451.176,A -85,B 0,C 180,E1 -15953.412,E2 -15953.412} C_VEL
LIN {X 0,Y 305.376,Z 441.57,A -85,B 0,C 180,E1 -15953.953,E2 -15953.953} C_VEL
LIN {X 0,Y 306.269,Z 434.725,A -85,B 0,C 180,E1 -15958.061,E2 -15958.061} C_VEL
LIN {X 0,Y 307.326,Z 427.833,A -85,B 0,C 180,E1 -15962.207,E2 -15962.207} C_VEL
LIN {X 0,Y 308.213,Z 422.389,A -85,B 0,C 180,E1 -15965.554,E2 -15965.554} C_VEL
LIN {X 0,Y 308.434,Z 419.902,A -85,B 0,C 180,E1 -15967.107,E2 -15967.107} C_VEL
LIN {X 0,Y 307.958,Z 416.003,A -85,B 0,C 180,E1 -15969.717,E2 -15969.717} C_VEL
LIN {X 0,Y 307.038,Z 410.962,A -85,B 0,C 180,E1 -15973.369,E2 -15973.369} C_VEL
LIN {X 0,Y 306.101,Z 405.914,A -85,B 0,C 180,E1 -15977.283,E2 -15977.283} C_VEL
LIN {X 0,Y 305.475,Z 402.436,A -85,B 0,C 180,E1 -15980.321,E2 -15980.321} C_VEL
LIN {X 0,Y 305.483,Z 402.432,A -85,B 0,C 180,E1 -15983.631,E2 -15983.631} C_VEL
LIN {X 0,Y 305.467,Z 402.435,A -85,B 0,C 180,E1 -15986.483,E2 -15986.483} C_VEL
LIN {X 0,Y 305.46,Z 402.434,A -85,B 0,C 180,E1 -15989.591,E2 -15989.591} C_VEL
LIN {X 0,Y 305.521,Z 402.43,A -85,B 0,C 180,E1 -15992.609,E2 -15992.609} C_VEL
LIN {X 0,Y 305.51,Z 402.427,A -85,B 0,C 180,E1 -15995.539,E2 -15995.539} C_VEL
LIN {X 0,Y 305.522,Z 402.426,A -85,B 0,C 180,E1 -15999.815,E2 -15999.815} C_VEL
LIN {X 0,Y 305.577,Z 402.423,A -85,B 0,C 180,E1 -16002.603,E2 -16002.603} C_VEL
LIN {X 0,Y 305.652,Z 402.41,A -85,B 0,C 180,E1 -16005.349,E2 -16005.349} C_VEL
LIN {X 0,Y 305.643,Z 402.411,A -85,B 0,C 180,E1 -16009.4,E2 -16009.4} C_VEL
LIN {X 0,Y 305.816,Z 402.391,A -85,B 0,C 180,E1 -16012.074,E2 -16012.074} C_VEL
LIN {X 0,Y 305.691,Z 402.408,A -85,B 0,C 180,E1 -16014.724,E2 -16014.724} C_VEL
LIN {X 0,Y 305.96,Z 402.373,A -85,B 0,C 180,E1 -16018.684,E2 -16018.684} C_VEL
LIN {X 0,Y 305.96,Z 402.37,A -85,B 0,C 180,E1 -16021.316,E2 -16021.316} C_VEL
LIN {X 0,Y 305.853,Z 402.385,A -85,B 0,C 180,E1 -16026.629,E2 -16026.629} C_VEL
LIN {X 0,Y 305.738,Z 402.398,A -85,B 0,C 180,E1 -16029.26,E2 -16029.26} C_VEL
LIN {X 0,Y 305.591,Z 402.416,A -85,B 0,C 180,E1 -16033.296,E2 -16033.296} C_VEL
LIN {X 0,Y 305.596,Z 402.42,A -85,B 0,C 180,E1 -16036.02,E2 -16036.02} C_VEL
LIN {X 0,Y 305.578,Z 402.418,A -85,B 0,C 180,E1 -16039.444,E2 -16039.444} C_VEL
LIN {X 0,Y 305.488,Z 402.43,A -85,B 0,C 180,E1 -16043.039,E2 -16043.039} C_VEL
LIN {X 0,Y 305.533,Z 402.426,A -85,B 0,C 180,E1 -16046.221,E2 -16046.221} C_VEL
LIN {X 0,Y 305.49,Z 402.429,A -85,B 0,C 180,E1 -16049.047,E2 -16049.047} C_VEL
LIN {X 0,Y 305.445,Z 402.437,A -85,B 0,C 180,E1 -16051.952,E2 -16051.952} C_VEL
LIN {X 0,Y 305.465,Z 402.433,A -85,B 0,C 180,E1 -16055.113,E2 -16055.113} C_VEL
LIN {X 0,Y 305.47,Z 402.432,A -85,B 0,C 180,E1 -16058.533,E2 -16058.533} C_VEL
LIN {X 0,Y 305.465,Z 402.432,A -85,B 0,C 180,E1 -16062.588,E2 -16062.588} C_VEL
LIN {X 0,Y 305.495,Z 402.43,A -85,B 0,C 180,E1 -16066.357,E2 -16066.357} C_VEL
LIN {X 0,Y 305.485,Z 402.434,A -85,B 0,C 180,E1 -16069.896,E2 -16069.896} C_VEL
LIN {X 0,Y 305.396,Z 402.446,A -85,B 0,C 180,E1 -16073.249,E2 -16073.249} C_VEL
LIN {X 0,Y 305.131,Z 402.481,A -85,B 0,C 180,E1 -16076.442,E2 -16076.442} C_VEL
LIN {X 0,Y 305.009,Z 403.219,A -85,B 0,C 180,E1 -16078.491,E2 -16078.491} C_VEL
LIN {X 0,Y 304.828,Z 406.443,A -85,B 0,C 180,E1 -16082.541,E2 -16082.541} C_VEL
LIN {X 0,Y 304.742,Z 409.507,A -85,B 0,C 180,E1 -16086.101,E2 -16086.101} C_VEL
LIN {X 0,Y 308.968,Z 422.401,A -85,B 0,C 180,E1 -16087.058,E2 -16087.058} C_VEL
LIN {X 0,Y 312.03,Z 433.768,A -85,B 0,C 180,E1 -16088.078,E2 -16088.078} C_VEL
LIN {X 0,Y 314.126,Z 444.494,A -85,B 0,C 180,E1 -16089.196,E2 -16089.196} C_VEL
LIN {X 0,Y 312.898,Z 455.209,A -85,B 0,C 180,E1 -16090.311,E2 -16090.311} C_VEL
LIN {X 0,Y 311.697,Z 465.049,A -85,B 0,C 180,E1 -16091.599,E2 -16091.599} C_VEL
LIN {X 0,Y 310.16,Z 474.982,A -85,B 0,C 180,E1 -16093.208,E2 -16093.208} C_VEL
LIN {X 0,Y 308.814,Z 483.108,A -85,B 0,C 180,E1 -16094.828,E2 -16094.828} C_VEL
LIN {X 0,Y 307.512,Z 491.06,A -85,B 0,C 180,E1 -16096.789,E2 -16096.789} C_VEL
LIN {X 0,Y 306.342,Z 497.443,A -85,B 0,C 180,E1 -16098.755,E2 -16098.755} C_VEL
LIN {X 0,Y 305.487,Z 502.498,A -85,B 0,C 180,E1 -16100.733,E2 -16100.733} C_VEL
LIN {X 0,Y 304.822,Z 506.675,A -85,B 0,C 180,E1 -16102.875,E2 -16102.875} C_VEL
LIN {X 0,Y 304.373,Z 509.317,A -85,B 0,C 180,E1 -16104.701,E2 -16104.701} C_VEL
LIN {X 0,Y 304.223,Z 510.699,A -85,B 0,C 180,E1 -16106.026,E2 -16106.026} C_VEL
LIN {X 0,Y 304.15,Z 511.679,A -85,B 0,C 180,E1 -16107.351,E2 -16107.351} C_VEL
LIN {X 0,Y 304.01,Z 512.516,A -85,B 0,C 180,E1 -16110,E2 -16110} C_VEL
LIN {X 0,Y 304.13,Z 511.743,A -85,B 0,C 180,E1 -16112.649,E2 -16112.649} C_VEL
LIN {X 0,Y 304.371,Z 509.443,A -85,B 0,C 180,E1 -16115.3,E2 -16115.3} C_VEL
LIN {X 0,Y 304.934,Z 505.92,A -85,B 0,C 180,E1 -16117.67,E2 -16117.67} C_VEL
LIN {X 0,Y 305.686,Z 501.185,A -85,B 0,C 180,E1 -16119.929,E2 -16119.929} C_VEL
LIN {X 0,Y 306.875,Z 494.779,A -85,B 0,C 180,E1 -16122.231,E2 -16122.231} C_VEL
LIN {X 0,Y 308.058,Z 487.738,A -85,B 0,C 180,E1 -16124.197,E2 -16124.197} C_VEL
LIN {X 0,Y 309.602,Z 478.953,A -85,B 0,C 180,E1 -16126.146,E2 -16126.146} C_VEL
LIN {X 0,Y 311.037,Z 469.935,A -85,B 0,C 180,E1 -16127.761,E2 -16127.761} C_VEL
LIN {X 0,Y 312.368,Z 459.517,A -85,B 0,C 180,E1 -16129.268,E2 -16129.268} C_VEL
LIN {X 0,Y 313.659,Z 448.821,A -85,B 0,C 180,E1 -16130.494,E2 -16130.494} C_VEL
LIN {X 0,Y 314.108,Z 443.877,A -85,B 0,C 180,E1 -16130.977,E2 -16130.977} C_VEL
LIN {X 0,Y 311.66,Z 432.221,A -85,B 0,C 180,E1 -16132.185,E2 -16132.185} C_VEL
LIN {X 0,Y 308.17,Z 419.763,A -85,B 0,C 180,E1 -16133.271,E2 -16133.271} C_VEL
LIN {X 0,Y 304.727,Z 409.43,A -85,B 0,C 180,E1 -16134.04,E2 -16134.04} C_VEL
LIN {X 0,Y 304.829,Z 406.54,A -85,B 0,C 180,E1 -16137.459,E2 -16137.459} C_VEL
LIN {X 0,Y 304.992,Z 404.128,A -85,B 0,C 180,E1 -16140.461,E2 -16140.461} C_VEL
LIN {X 0,Y 305.011,Z 402.949,A -85,B 0,C 180,E1 -16142.003,E2 -16142.003} C_VEL
LIN {X 0,Y 305.186,Z 402.471,A -85,B 0,C 180,E1 -16144.001,E2 -16144.001} C_VEL
LIN {X 0,Y 305.392,Z 402.446,A -85,B 0,C 180,E1 -16146.751,E2 -16146.751} C_VEL
LIN {X 0,Y 305.46,Z 402.436,A -85,B 0,C 180,E1 -16150.108,E2 -16150.108} C_VEL
LIN {X 0,Y 305.428,Z 402.437,A -85,B 0,C 180,E1 -16153.655,E2 -16153.655} C_VEL
LIN {X 0,Y 305.458,Z 402.433,A -85,B 0,C 180,E1 -16157.414,E2 -16157.414} C_VEL
LIN {X 0,Y 305.499,Z 402.427,A -85,B 0,C 180,E1 -16161.601,E2 -16161.601} C_VEL
LIN {X 0,Y 305.466,Z 402.432,A -85,B 0,C 180,E1 -16164.887,E2 -16164.887} C_VEL
LIN {X 0,Y 305.454,Z 402.438,A -85,B 0,C 180,E1 -16168.355,E2 -16168.355} C_VEL
LIN {X 0,Y 305.516,Z 402.426,A -85,B 0,C 180,E1 -16171.113,E2 -16171.113} C_VEL
LIN {X 0,Y 305.574,Z 402.424,A -85,B 0,C 180,E1 -16174.088,E2 -16174.088} C_VEL
LIN {X 0,Y 305.485,Z 402.432,A -85,B 0,C 180,E1 -16178.402,E2 -16178.402} C_VEL
LIN {X 0,Y 305.593,Z 402.416,A -85,B 0,C 180,E1 -16181.218,E2 -16181.218} C_VEL
LIN {X 0,Y 305.636,Z 402.411,A -85,B 0,C 180,E1 -16184.896,E2 -16184.896} C_VEL
LIN {X 0,Y 305.019,Z 402.491,A -85,B 0,C 180,E1 -16185.995,E2 -16185.995} C_VEL
LIN {X 0,Y 302.129,Z 402.852,A -85,B 0,C 180,E1 -16187.784,E2 -16187.784} C_VEL
LIN {X 0,Y 299.685,Z 403.155,A -85,B 0,C 180,E1 -16189.235,E2 -16189.235} C_VEL
LIN {X 0,Y 298.701,Z 403.278,A -85,B 0,C 180,E1 -16190.36,E2 -16190.36} C_VEL
LIN {X 0,Y 298.659,Z 403.281,A -85,B 0,C 180,E1 -16190.741,E2 -16190.741} C_VEL
LIN {X 0,Y 298.781,Z 403.266,A -85,B 0,C 180,E1 -16193.246,E2 -16193.246} C_VEL
LIN {X 0,Y 298.926,Z 403.248,A -85,B 0,C 180,E1 -16198.653,E2 -16198.653} C_VEL
LIN {X 0,Y 298.926,Z 403.251,A -85,B 0,C 180,E1 -16201.347,E2 -16201.347} C_VEL
LIN {X 0,Y 298.802,Z 403.263,A -85,B 0,C 180,E1 -16206.754,E2 -16206.754} C_VEL
LIN {X 0,Y 298.685,Z 403.282,A -85,B 0,C 180,E1 -16209.48,E2 -16209.48} C_VEL
LIN {X 0,Y 298.558,Z 403.296,A -85,B 0,C 180,E1 -16213.615,E2 -16213.615} C_VEL
LIN {X 0,Y 298.553,Z 403.293,A -85,B 0,C 180,E1 -16216.408,E2 -16216.408} C_VEL
LIN {X 0,Y 298.515,Z 403.301,A -85,B 0,C 180,E1 -16219.655,E2 -16219.655} C_VEL
LIN {X 0,Y 298.461,Z 403.309,A -85,B 0,C 180,E1 -16223.597,E2 -16223.597} C_VEL
LIN {X 0,Y 298.49,Z 403.303,A -85,B 0,C 180,E1 -16226.574,E2 -16226.574} C_VEL
LIN {X 0,Y 298.42,Z 403.314,A -85,B 0,C 180,E1 -16229.641,E2 -16229.641} C_VEL
LIN {X 0,Y 298.398,Z 403.316,A -85,B 0,C 180,E1 -16232.8,E2 -16232.8} C_VEL
LIN {X 0,Y 298.449,Z 403.311,A -85,B 0,C 180,E1 -16236.807,E2 -16236.807} C_VEL
LIN {X 0,Y 298.434,Z 403.371,A -85,B 0,C 180,E1 -16239.181,E2 -16239.181} C_VEL
LIN {X 0,Y 299.322,Z 408.155,A -85,B 0,C 180,E1 -16243.291,E2 -16243.291} C_VEL
LIN {X 0,Y 300.24,Z 413.219,A -85,B 0,C 180,E1 -16247.247,E2 -16247.247} C_VEL
LIN {X 0,Y 301.117,Z 418.265,A -85,B 0,C 180,E1 -16250.937,E2 -16250.937} C_VEL
LIN {X 0,Y 301.327,Z 422.055,A -85,B 0,C 180,E1 -16253.505,E2 -16253.505} C_VEL
LIN {X 0,Y 300.582,Z 427.007,A -85,B 0,C 180,E1 -16256.67,E2 -16256.67} C_VEL
LIN {X 0,Y 299.574,Z 433.127,A -85,B 0,C 180,E1 -16260.484,E2 -16260.484} C_VEL
LIN {X 0,Y 298.697,Z 439.149,A -85,B 0,C 180,E1 -16264.196,E2 -16264.196} C_VEL
LIN {X 0,Y 298.427,Z 441.162,A -85,B 0,C 180,E1 -16265.433,E2 -16265.433} C_VEL
LIN {X 0,Y 301.29,Z 454.63,A -85,B 0,C 180,E1 -16266.259,E2 -16266.259} C_VEL
LIN {X 0,Y 303.15,Z 467.18,A -85,B 0,C 180,E1 -16267.235,E2 -16267.235} C_VEL
LIN {X 0,Y 304.191,Z 478.468,A -85,B 0,C 180,E1 -16268.305,E2 -16268.305} C_VEL
LIN {X 0,Y 304.811,Z 489.639,A -85,B 0,C 180,E1 -16269.59,E2 -16269.59} C_VEL
LIN {X 0,Y 303.102,Z 500.917,A -85,B 0,C 180,E1 -16271.057,E2 -16271.057} C_VEL
LIN {X 0,Y 301.496,Z 510.998,A -85,B 0,C 180,E1 -16272.725,E2 -16272.725} C_VEL
LIN {X 0,Y 300.293,Z 519.142,A -85,B 0,C 180,E1 -16274.386,E2 -16274.386} C_VEL
LIN {X 0,Y 298.928,Z 527.208,A -85,B 0,C 180,E1 -16276.402,E2 -16276.402} C_VEL
LIN {X 0,Y 297.91,Z 533.687,A -85,B 0,C 180,E1 -16278.432,E2 -16278.432} C_VEL
LIN {X 0,Y 297.273,Z 538.847,A -85,B 0,C 180,E1 -16280.474,E2 -16280.474} C_VEL
LIN {X 0,Y 296.869,Z 542.86,A -85,B 0,C 180,E1 -16282.518,E2 -16282.518} C_VEL
LIN {X 0,Y 296.689,Z 545.832,A -85,B 0,C 180,E1 -16284.563,E2 -16284.563} C_VEL
LIN {X 0,Y 296.667,Z 547.25,A -85,B 0,C 180,E1 -16285.924,E2 -16285.924} C_VEL
LIN {X 0,Y 296.639,Z 548.262,A -85,B 0,C 180,E1 -16287.284,E2 -16287.284} C_VEL
LIN {X 0,Y 296.674,Z 548.882,A -85,B 0,C 180,E1 -16288.642,E2 -16288.642} C_VEL
LIN {X 0,Y 296.782,Z 549.106,A -85,B 0,C 180,E1 -16290,E2 -16290} C_VEL
LIN {X 0,Y 296.696,Z 548.879,A -85,B 0,C 180,E1 -16291.357,E2 -16291.357} C_VEL
LIN {X 0,Y 296.667,Z 547.243,A -85,B 0,C 180,E1 -16294.075,E2 -16294.075} C_VEL
LIN {X 0,Y 296.738,Z 545.235,A -85,B 0,C 180,E1 -16295.88,E2 -16295.88} C_VEL
LIN {X 0,Y 296.963,Z 541.595,A -85,B 0,C 180,E1 -16298.163,E2 -16298.163} C_VEL
LIN {X 0,Y 297.458,Z 537.205,A -85,B 0,C 180,E1 -16300.207,E2 -16300.207} C_VEL
LIN {X 0,Y 298.179,Z 531.619,A -85,B 0,C 180,E1 -16302.247,E2 -16302.247} C_VEL
LIN {X 0,Y 299.379,Z 524.671,A -85,B 0,C 180,E1 -16304.27,E2 -16304.27} C_VEL
LIN {X 0,Y 300.567,Z 517.582,A -85,B 0,C 180,E1 -16305.947,E2 -16305.947} C_VEL
LIN {X 0,Y 301.786,Z 509.033,A -85,B 0,C 180,E1 -16307.623,E2 -16307.623} C_VEL
LIN {X 0,Y 303.491,Z 498.499,A -85,B 0,C 180,E1 -16309.268,E2 -16309.268} C_VEL
LIN {X 0,Y 304.76,Z 489.513,A -85,B 0,C 180,E1 -16310.414,E2 -16310.414} C_VEL
LIN {X 0,Y 304.185,Z 478.307,A -85,B 0,C 180,E1 -16311.695,E2 -16311.695} C_VEL
LIN {X 0,Y 303.002,Z 466.083,A -85,B 0,C 180,E1 -16312.845,E2 -16312.845} C_VEL
LIN {X 0,Y 300.968,Z 453.113,A -85,B 0,C 180,E1 -16313.827,E2 -16313.827} C_VEL
LIN {X 0,Y 298.441,Z 441.097,A -85,B 0,C 180,E1 -16314.552,E2 -16314.552} C_VEL
LIN {X 0,Y 299.387,Z 434.31,A -85,B 0,C 180,E1 -16318.766,E2 -16318.766} C_VEL
LIN {X 0,Y 300.375,Z 428.112,A -85,B 0,C 180,E1 -16322.615,E2 -16322.615} C_VEL
LIN {X 0,Y 301.22,Z 423.265,A -85,B 0,C 180,E1 -16325.683,E2 -16325.683} C_VEL
LIN {X 0,Y 301.385,Z 420.402,A -85,B 0,C 180,E1 -16327.547,E2 -16327.547} C_VEL
LIN {X 0,Y 300.686,Z 415.631,A -85,B 0,C 180,E1 -16330.878,E2 -16330.878} C_VEL
LIN {X 0,Y 299.765,Z 410.592,A -85,B 0,C 180,E1 -16334.697,E2 -16334.697} C_VEL
LIN {X 0,Y 298.836,Z 405.61,A -85,B 0,C 180,E1 -16338.814,E2 -16338.814} C_VEL
LIN {X 0,Y 298.428,Z 403.312,A -85,B 0,C 180,E1 -16341.001,E2 -16341.001} C_VEL
LIN {X 0,Y 298.421,Z 403.312,A -85,B 0,C 180,E1 -16343.93,E2 -16343.93} C_VEL
LIN {X 0,Y 298.396,Z 403.316,A -85,B 0,C 180,E1 -16347.984,E2 -16347.984} C_VEL
LIN {X 0,Y 298.461,Z 403.306,A -85,B 0,C 180,E1 -16351.904,E2 -16351.904} C_VEL
LIN {X 0,Y 298.487,Z 403.305,A -85,B 0,C 180,E1 -16354.924,E2 -16354.924} C_VEL
LIN {X 0,Y 298.453,Z 403.307,A -85,B 0,C 180,E1 -16359.315,E2 -16359.315} C_VEL
LIN {X 0,Y 298.54,Z 403.297,A -85,B 0,C 180,E1 -16362.18,E2 -16362.18} C_VEL
LIN {X 0,Y 298.596,Z 403.291,A -85,B 0,C 180,E1 -16364.995,E2 -16364.995} C_VEL
LIN {X 0,Y 298.598,Z 403.289,A -85,B 0,C 180,E1 -16369.147,E2 -16369.147} C_VEL
LIN {X 0,Y 298.761,Z 403.269,A -85,B 0,C 180,E1 -16371.886,E2 -16371.886} C_VEL
LIN {X 0,Y 298.663,Z 403.284,A -85,B 0,C 180,E1 -16374.599,E2 -16374.599} C_VEL
LIN {X 0,Y 298.926,Z 403.249,A -85,B 0,C 180,E1 -16378.653,E2 -16378.653} C_VEL
LIN {X 0,Y 298.926,Z 403.246,A -85,B 0,C 180,E1 -16381.347,E2 -16381.347} C_VEL
LIN {X 0,Y 298.801,Z 403.263,A -85,B 0,C 180,E1 -16386.754,E2 -16386.754} C_VEL
LIN {X 0,Y 298.683,Z 403.278,A -85,B 0,C 180,E1 -16389.48,E2 -16389.48} C_VEL
LIN {X 0,Y 298.555,Z 403.294,A -85,B 0,C 180,E1 -16393.615,E2 -16393.615} C_VEL
LIN {X 0,Y 298.551,Z 403.296,A -85,B 0,C 180,E1 -16396.409,E2 -16396.409} C_VEL
LIN {X 0,Y 298.512,Z 403.3,A -85,B 0,C 180,E1 -16399.654,E2 -16399.654} C_VEL
LIN {X 0,Y 298.431,Z 403.311,A -85,B 0,C 180,E1 -16403.6,E2 -16403.6} C_VEL
LIN {X 0,Y 298.488,Z 403.302,A -85,B 0,C 180,E1 -16406.575,E2 -16406.575} C_VEL
LIN {X 0,Y 298.419,Z 403.313,A -85,B 0,C 180,E1 -16409.641,E2 -16409.641} C_VEL
LIN {X 0,Y 298.397,Z 403.31,A -85,B 0,C 180,E1 -16412.8,E2 -16412.8} C_VEL
LIN {X 0,Y 298.467,Z 403.302,A -85,B 0,C 180,E1 -16416.813,E2 -16416.813} C_VEL
LIN {X 0,Y 298.39,Z 403.314,A -85,B 0,C 180,E1 -16421.088,E2 -16421.088} C_VEL
LIN {X 0,Y 298.418,Z 403.311,A -85,B 0,C 180,E1 -16424.953,E2 -16424.953} C_VEL
LIN {X 0,Y 298.454,Z 403.307,A -85,B 0,C 180,E1 -16428.75,E2 -16428.75} C_VEL
LIN {X 0,Y 298.399,Z 403.316,A -85,B 0,C 180,E1 -16432.239,E2 -16432.239} C_VEL
LIN {X 0,Y 298.16,Z 403.35,A -85,B 0,C 180,E1 -16435.588,E2 -16435.588} C_VEL
LIN {X 0,Y 297.988,Z 403.37,A -85,B 0,C 180,E1 -16437.149,E2 -16437.149} C_VEL
LIN {X 0,Y 297.881,Z 406.048,A -85,B 0,C 180,E1 -16440.804,E2 -16440.804} C_VEL
LIN {X 0,Y 297.727,Z 409.386,A -85,B 0,C 180,E1 -16444.856,E2 -16444.856} C_VEL
LIN {X 0,Y 297.718,Z 409.924,A -85,B 0,C 180,E1 -16445.495,E2 -16445.495} C_VEL
LIN {X 0,Y 302.087,Z 423.027,A -85,B 0,C 180,E1 -16446.514,E2 -16446.514} C_VEL
LIN {X 0,Y 305.127,Z 434.154,A -85,B 0,C 180,E1 -16447.549,E2 -16447.549} C_VEL
LIN {X 0,Y 307.355,Z 444.942,A -85,B 0,C 180,E1 -16448.715,E2 -16448.715} C_VEL
LIN {X 0,Y 306.243,Z 455.646,A -85,B 0,C 180,E1 -16449.865,E2 -16449.865} C_VEL
LIN {X 0,Y 304.978,Z 465.484,A -85,B 0,C 180,E1 -16451.179,E2 -16451.179} C_VEL
LIN {X 0,Y 303.397,Z 475.415,A -85,B 0,C 180,E1 -16452.822,E2 -16452.822} C_VEL
LIN {X 0,Y 301.985,Z 483.542,A -85,B 0,C 180,E1 -16454.476,E2 -16454.476} C_VEL
LIN {X 0,Y 300.614,Z 491.494,A -85,B 0,C 180,E1 -16456.48,E2 -16456.48} C_VEL
LIN {X 0,Y 299.415,Z 497.875,A -85,B 0,C 180,E1 -16458.491,E2 -16458.491} C_VEL
